(* CODESYS project TcNexaHmi.library
   Author: ATI Software Engineering
   Version: 2.0.0
   Title: TcNexaHmi
   DefaultNamespace: TcNexa_Devices_Hmi_TcNexaHmi
   Placeholder: TcNexaHmi
   Company: TcNexa

Project tree, tasks and I/O mapping:
  libraries: Tc2_Standard, * (Beckhoff Automation GmbH); Tc2_System, * (Beckhoff Automation GmbH); Tc2_Utilities, * (Beckhoff Automation GmbH); Tc3_IotBase, * (Beckhoff Automation GmbH); Tc3_Module, * (Beckhoff Automation GmbH); TcUtilities, * (TcNexa)
  Base/
    ITFs/
      interface I_NexaHmi: isConnected, messageFullTopic, messageLastTopicLevel, messagePayload, onNewMessage, publish, publishAdr, subscribe, topicPrefix, unsubscribe
    POUs/
      function block FB_NexaHmi [ST]: hostName, hostPort, id, isConnected, messageFullTopic, messageLastTopicLevel, messagePayload, onNewMessage, topicPrefix, FB_main, publish, publishAdr, setWill, subscribe, unsubscribe
    data type E_UserLevel
    function F_GetUserLevelAsString [ST]
  Device Buttons/
    function block FB_NexaHmiDeviceButton [ST]: _handleNewMessages, _onConnection, _updateTopics, FB_init, Buttons, description, FB_main
  Elements/
    Counters/
      data type E_NexaHmiCounterColor
      function block FB_NexaHmiCounter [ST]: color, description, name, value, _getColor, _handleNewMessages, _onConnection, _updateTopics, clear, FB_init, FB_main, inc
    Graph 2D/
      data type E_GraphLineColor2D
      function block FB_NexaHmi_Graph2D [ST]: _onConnection, _updateTopics, FB_init, description, Lines, xMax, xMaxVisible, xMin, xMinVisible, yMax, yMaxVisible, yMin, yMinVisible, clear, FB_main, publish
      function block FB_NexaHmi_GraphLine2D [ST]: _clearBuffer, _getColor, _onConnection, _updateTopics, Hmi, topicPrefix, addPoint, clear, FB_main, publish, setColor
    POUs/
      function block FB_CustomHmiButton [ST]: focused, name, onTap, visible, clear
      function block FB_GeneralHmiButton [ST]: confirmationRequired, enabled, focused, isPressed, loggingEnabled, name, onTap, visible, clear
      function block FB_ModeHmiButton [ST]: enabled, onLongPress, onTap, visible, clear, clearCommand
      function block FB_NexaHmiCustomButtons [ST]: Buttons, clear
      function block FB_NexaHmiTextFields [ST]: fields, userAction, clear
  GVLs/
    global variables GVL_TcNexaHmiUtilities
  Order/
    function block FB_NexaHmiOrderBOOL [ST]: _handleNewMessages, _onConnection, _updateTopics, FB_init, description, name, value, FB_main
    function block FB_NexaHmiOrderINT [ST]: _handleNewMessage, _onConnection, _updateTopics, FB_init, description, lowerLimit, name, upperLimit, value, FB_main
    function block FB_NexaHmiOrderREAL [ST]: _handleNewMessage, _onConnection, _updateTopics, FB_init, description, lowerLimit, name, upperLimit, value, FB_main
    function block FB_NexaHmiOrderSTRING [ST]: _handleNewMessages, _onConnection, _updateTopics, FB_init, value, FB_main
    function block FB_NexaHmiOrderTIME [ST]: _handleNewMessages, _onConnection, _updateTopics, FB_init, description, name, value, FB_main
  Persistent/
    function block FB_NexaHmiPersistentBase [ST]: _handleVar, _onConnection, FB_init, FB_main
    function block FB_NexaHmiPersistentBOOL [ST]: _handleVar, FB_init, value
    function block FB_NexaHmiPersistentINT [ST]: _handleVar, FB_init, value
    function block FB_NexaHmiPersistentREAL [ST]: _handleVar, FB_init, value
    function block FB_NexaHmiPersistentSTRING [ST]: _handleVar, FB_init, value
    function block FB_NexaHmiPersistentTIME [ST]: _handleVar, FB_init, value
    function block FB_NexaHmiPersistentXYZ [ST]: _handleVar, FB_init, velocity, X, Y, Z
  Settings/
    function block FB_NexaHmiSettingBase [ST]: _handleVars, _onConnection, _updateTopics, FB_init, description, enabled, name, userLevel, FB_main
    function block FB_NexaHmiSettingBOOL [ST]: _handleVars, FB_init, value
    function block FB_NexaHmiSettingCHOICE [ST]: _handleVars, FB_init, value
    function block FB_NexaHmiSettingINT [ST]: _handleVars, FB_init, lowerLimit, upperLimit, value
    function block FB_NexaHmiSettingREAL [ST]: _handleVars, FB_init, lowerLimit, upperLimit, value
    function block FB_NexaHmiSettingSTRING [ST]: _handleVars, FB_init, value
    function block FB_NexaHmiSettingTIME [ST]: _handleVars, FB_init, lowerLimit, upperLimit, value
  Tests/
    program PRG_TEST [ST]
  Version/
    global variables Global_Version
*)

// Base/E_UserLevel
{attribute 'qualified_only'}
{attribute 'strict'}
TYPE E_UserLevel :
(
	Operator := 0,
	LineLeader,
	Maintenance,
	Administrator,
	System
):= Administrator;
END_TYPE

// Elements/Counters/E_NexaHmiCounterColor
{attribute 'qualified_only'}
{attribute 'strict'}
TYPE E_NexaHmiCounterColor :
(
	black := 0,
	red,
	blue,
	green,
	yellow,
	purple,
	grey
):= black;
END_TYPE

// Elements/Graph 2D/E_GraphLineColor2D
{attribute 'qualified_only'}
{attribute 'strict'}
TYPE E_GraphLineColor2D :
(
	black := 0,
	red,
	blue,
	green,
	yellow,
	purple,
	grey
):= black;
END_TYPE

// GVLs/GVL_TcNexaHmiUtilities
{attribute 'qualified_only'}
VAR_GLOBAL CONSTANT
	numOfTextFields			: USINT:= 3;
	numOfCustomButtons		: USINT:= 5;
	numOfGraphLines2D		: USINT:= 5;
END_VAR

// Version/Global_Version
{attribute 'TcGenerated'}
{attribute 'no-analysis'}
{attribute 'linkalways'}
// This function has been automatically generated from the project information.
VAR_GLOBAL CONSTANT
	{attribute 'const_non_replaced'}
	stLibVersion_TcNexaHmi : ST_LibVersion := (iMajor := 2, iMinor := 0, iBuild := 0, iRevision := 0, nFlags := 0, sVersion := '2.0.0');
END_VAR

// Base/ITFs/I_NexaHmi
INTERFACE I_NexaHmi

PROPERTY PUBLIC isConnected : BOOL
GET
END_GET
END_PROPERTY

PROPERTY messageFullTopic : Tc2_System.T_MaxString
GET
END_GET
END_PROPERTY

PROPERTY PUBLIC messageLastTopicLevel : STRING
GET
END_GET
END_PROPERTY

PROPERTY messagePayload : Tc2_System.T_MaxString
GET
END_GET
END_PROPERTY

PROPERTY PUBLIC onNewMessage : BOOL
GET
END_GET
END_PROPERTY

METHOD PUBLIC publish : BOOL
VAR_INPUT
	topic		: Tc2_System.T_MaxString;
	payload		: Tc2_System.T_MaxString;
END_VAR
END_METHOD

METHOD PUBLIC publishAdr : BOOL
VAR_INPUT
	topic		: Tc2_System.T_MaxString;
	payload		: PVOID;
	payloadSize	: UDINT;
END_VAR
END_METHOD

METHOD PUBLIC subscribe : BOOL
VAR_INPUT
	topic		: Tc2_System.T_MaxString;
END_VAR
END_METHOD

PROPERTY PUBLIC topicPrefix : Tc2_System.T_MaxString
GET
END_GET
END_PROPERTY

METHOD PUBLIC unsubscribe
VAR_INPUT
	topic		: Tc2_System.T_MaxString;
END_VAR
END_METHOD

END_INTERFACE

// Base/POUs/FB_NexaHmi
FUNCTION_BLOCK FB_NexaHmi IMPLEMENTS I_NexaHmi
VAR
	(* Mqtt *)
	_Client						: Tc3_IotBase.FB_IotMqttClient;
	_ClientMessageQueue			: Tc3_IotBase.FB_IotMqttMessageQueue;
	_ClientMessage				: Tc3_IotBase.FB_IotMqttMessage;
	_isInit						: BOOL;
	_onNewMessage				: BOOL;
	_topicPrefix				: Tc2_System.T_MaxString;
	(* Message *)
	_messageTopic				: Tc2_System.T_MaxString;
	_messageTopicSplitter		: TcNexa_Components_TcUtilities.FB_TextSplitter;
	_messagePayload				: Tc2_System.T_MaxString;
	(* Will *)
	_willTopic					: STRING;
	_willPayload				: STRING;
END_VAR

PROPERTY PUBLIC hostName : Tc2_System.T_MaxString
GET
hostName:= _Client.sHostName;
END_GET
SET
_Client.sHostName:= hostName;
END_SET
END_PROPERTY

PROPERTY PUBLIC hostPort : UINT
GET
hostPort:= _Client.nHostPort;
END_GET
SET
_Client.nHostPort:= hostPort;
END_SET
END_PROPERTY

PROPERTY PUBLIC id : Tc2_System.T_MaxString
GET
id:= _Client.sClientId;
END_GET
SET
_Client.sClientId:= id;
END_SET
END_PROPERTY

PROPERTY PUBLIC isConnected : BOOL
GET
isConnected:= _Client.bConnected;
END_GET
END_PROPERTY

PROPERTY messageFullTopic : Tc2_System.T_MaxString
GET
messageFullTopic:= _messageTopic;
END_GET
END_PROPERTY

PROPERTY PUBLIC messageLastTopicLevel : STRING
GET
messageLastTopicLevel:= _messageTopicSplitter.getValueAt(index:= _messageTopicSplitter.size, Response:= 0);
END_GET
END_PROPERTY

PROPERTY messagePayload : Tc2_System.T_MaxString
GET
messagePayload:= _messagePayload;
END_GET
END_PROPERTY

PROPERTY PUBLIC onNewMessage : BOOL
GET
onNewMessage:= _onNewMessage;
END_GET
END_PROPERTY

PROPERTY PUBLIC topicPrefix : Tc2_System.T_MaxString
GET
topicPrefix:= _topicPrefix;
END_GET
SET
_topicPrefix:= topicPrefix;
END_SET
END_PROPERTY

METHOD PUBLIC FB_main
VAR_INPUT
END_VAR
IF NOT _isInit THEN
	_Client.ipMessageQueue:= _ClientMessageQueue;
	_isInit:= TRUE;
END_IF
_Client.Execute(bConnect:= TRUE);

_onNewMessage:= FALSE;
IF (_ClientMessageQueue.nQueuedMessages > 0) THEN
	IF _ClientMessageQueue.Dequeue(fbMessage:= _ClientMessage)  THEN
		_ClientMessage.GetTopic(
			pTopic				:= ADR(_messageTopic),
			nTopicSize			:= SIZEOF(_messageTopic));
		_ClientMessage.GetPayload(
			pPayload			:= ADR(_messagePayload),
			nPayloadSize		:= SIZEOF(_messagePayload),
			bSetNullTermination	:= TRUE);
		_messageTopicSplitter.split(
			source				:= _messageTopic,
			delimiter			:= '/',
			Response			:= 0);
		_onNewMessage:= TRUE;
	END_IF
ELSE
	_messageTopic:= '';
	_messagePayload:= '';
END_IF
END_METHOD

METHOD PUBLIC publish : BOOL
VAR_INPUT
	topic		: Tc2_System.T_MaxString;
	payload		: Tc2_System.T_MaxString;
END_VAR
publish:= _Client.Publish(
			sTopic			:= topic,
			pPayload		:= ADR(payload),
			nPayloadSize	:= INT_TO_UDINT(Tc2_Standard.LEN(payload)),
			eQoS			:= TcIotMqttQos.AtMostOnceDelivery,
			bRetain			:= TRUE,
			bQueue			:= FALSE);
END_METHOD

METHOD PUBLIC publishAdr : BOOL
VAR_INPUT
	topic		: Tc2_System.T_MaxString;
	payload		: PVOID;
	payloadSize	: UDINT;
END_VAR
publishAdr:= _Client.Publish(
			sTopic			:= topic,
			pPayload		:= payload,
			nPayloadSize	:= payloadSize,
			eQoS			:= TcIotMqttQos.AtMostOnceDelivery,
			bRetain			:= TRUE,
			bQueue			:= FALSE);
END_METHOD

METHOD PUBLIC setWill
VAR_INPUT
	topic		: Tc2_System.T_MaxString;
	payload		: Tc2_System.T_MaxString;
END_VAR
_willTopic:= topic;
THIS^._willPayload:= payload;
THIS^._Client.stWill.sTopic:= _willTopic;
THIS^._Client.stWill.pPayload:= ADR(_willPayload);
THIS^._Client.stWill.nPayloadSize:= INT_TO_UDINT(Tc2_Standard.LEN(_willPayload));
THIS^._Client.stWill.eQoS:= TcIotMqttQos.AtMostOnceDelivery;
THIS^._Client.stWill.bRetain:= TRUE;
END_METHOD

METHOD PUBLIC subscribe : BOOL
VAR_INPUT
	topic		: Tc2_System.T_MaxString;
END_VAR
subscribe:= _Client.Subscribe(
				sTopic	:= topic,
				eQoS	:= TcIotMqttQos.AtLeastOnceDelivery);
END_METHOD

METHOD PUBLIC unsubscribe
VAR_INPUT
	topic		: Tc2_System.T_MaxString;
END_VAR
_Client.Unsubscribe(sTopic:= topic);
END_METHOD

END_FUNCTION_BLOCK

// Base/F_GetUserLevelAsString
FUNCTION F_GetUserLevelAsString : STRING
VAR_INPUT
	userLevel		: E_UserLevel;
END_VAR
VAR
END_VAR

IF (userLevel = E_UserLevel.Operator) THEN
	F_GetUserLevelAsString:= 'operator';
ELSIF (userLevel = E_UserLevel.LineLeader) THEN
	F_GetUserLevelAsString:= 'lineLeader';
ELSIF (userLevel = E_UserLevel.Maintenance) THEN
	F_GetUserLevelAsString:= 'maintenance';
ELSIF (userLevel = E_UserLevel.Administrator) THEN
	F_GetUserLevelAsString:= 'admin';
ELSIF (userLevel = E_UserLevel.System) THEN
	F_GetUserLevelAsString:= 'system';
END_IF

END_FUNCTION

// Device Buttons/FB_NexaHmiDeviceButton
FUNCTION_BLOCK FB_NexaHmiDeviceButton
VAR
	_Hmi				: I_NexaHmi;
	_timerConnected		: Tc2_Standard.TON;
	_onHmiConnection	: Tc2_Standard.R_TRIG;
	_isHmiConnected		: BOOL;
	_topicPrefix		: Tc2_System.T_MaxString;
	_id					: UINT;
	_name				: Tc2_System.T_MaxString;
	_description		: Tc2_System.T_MaxString;
	_Buttons			: ARRAY[1..NUM_OF_BUTTONS] OF FB_GeneralHmiButton;
	_LastButtons		: ARRAY[1..NUM_OF_BUTTONS] OF FB_GeneralHmiButton;
	_lastDescription	: Tc2_System.T_MaxString;		
	_tmpCounter			: USINT;
	_tmpText			: Tc2_System.T_MaxString;
END_VAR
VAR CONSTANT
	NUM_OF_BUTTONS		: USINT:= 3;
END_VAR

METHOD PROTECTED _handleNewMessages
VAR_INPUT
END_VAR
IF NOT _isHmiConnected THEN RETURN; END_IF

IF _Hmi.onNewMessage THEN
	FOR _tmpCounter:= 1 TO NUM_OF_BUTTONS DO
		_tmpText:= Tc2_Standard.CONCAT(STR1:= _topicPrefix, STR2:= 'buttons/');
		_tmpText:= Tc2_Standard.CONCAT(STR1:= _tmpText, STR2:= USINT_TO_STRING(_tmpCounter));
		_tmpText:= Tc2_Standard.CONCAT(STR1:= _tmpText, STR2:= '/action');
		IF (_Hmi.messageFullTopic = _tmpText) THEN
			IF (_Hmi.messagePayload = 'tap') AND _Buttons[_tmpCounter].enabled THEN
				_Buttons[_tmpCounter].onTap:= TRUE;
// 			ELSIF (_Hmi.messagePayload = 'longPress') AND _Buttons[_tmpCounter].enabled THEN
// 				_Buttons[_tmpCounter].isPressed:= TRUE;
			END_IF
		END_IF
	END_FOR
END_IF
END_METHOD

METHOD PROTECTED _onConnection
VAR_INPUT
END_VAR
IF NOT _onHmiConnection.Q THEN RETURN; END_IF

_topicPrefix:= Tc2_Standard.CONCAT(STR1:= _Hmi.topicPrefix, STR2:= 'devices/buttons/');
_topicPrefix:= Tc2_Standard.CONCAT(STR1:= _topicPrefix, STR2:= UINT_TO_STRING(_id));
_topicPrefix:= Tc2_Standard.CONCAT(STR1:= _topicPrefix, STR2:= '/');

FOR _tmpCounter:= 1 TO NUM_OF_BUTTONS DO
	_tmpText:= CONCAT(STR1:= _topicPrefix, STR2:= 'buttons/');
	_tmpText:= CONCAT(STR1:= _tmpText, STR2:= USINT_TO_STRING(_tmpCounter));
	_tmpText:= CONCAT(STR1:= _tmpText, STR2:= '/action');
	_Hmi.subscribe(topic:= _tmpText);
END_FOR

_Hmi.publish(
	topic	:= Tc2_Standard.CONCAT(STR1:= _topicPrefix, STR2:= 'active'),
	payload	:= BOOL_TO_STRING(TRUE));
_Hmi.publish(
	topic	:= Tc2_Standard.CONCAT(STR1:= _topicPrefix, STR2:= 'name'),
	payload	:= _name);
END_METHOD

METHOD PROTECTED _updateTopics
VAR_INPUT
END_VAR
IF NOT _isHmiConnected THEN RETURN; END_IF

(* Description *)
IF (_lastDescription <> _description) OR _onHmiConnection.Q THEN
	_lastDescription:= _description;
	_Hmi.publish(
		topic	:= Tc2_Standard.CONCAT(STR1:= _topicPrefix, STR2:= 'description'),
		payload	:= _description);
END_IF
(* Handle Buttons *)
FOR _tmpCounter:= 1 TO NUM_OF_BUTTONS DO
	(* Button Name *)
	IF (_LastButtons[_tmpCounter].name <> _Buttons[_tmpCounter].name) OR _onHmiConnection.Q THEN
		_LastButtons[_tmpCounter].name:= _Buttons[_tmpCounter].name;
		_tmpText:= Tc2_Standard.CONCAT(STR1:= _topicPrefix, STR2:= 'buttons/');
		_tmpText:= Tc2_Standard.CONCAT(STR1:= _tmpText, STR2:= USINT_TO_STRING(_tmpCounter));
		_tmpText:= Tc2_Standard.CONCAT(STR1:= _tmpText, STR2:= '/name');
		_Hmi.publish(
			topic	:= _tmpText,
			payload	:= _Buttons[_tmpCounter].name);
	END_IF
	(* Button Visible *)
	IF (_LastButtons[_tmpCounter].visible <> _Buttons[_tmpCounter].visible) OR _onHmiConnection.Q THEN
		_LastButtons[_tmpCounter].visible:= _Buttons[_tmpCounter].visible;
		_tmpText:= Tc2_Standard.CONCAT(STR1:= _topicPrefix, STR2:= 'buttons/');
		_tmpText:= Tc2_Standard.CONCAT(STR1:= _tmpText, STR2:= USINT_TO_STRING(_tmpCounter));
		_tmpText:= Tc2_Standard.CONCAT(STR1:= _tmpText, STR2:= '/visible');
		_Hmi.publish(
			topic	:= _tmpText,
			payload	:= BOOL_TO_STRING(_Buttons[_tmpCounter].visible));
	END_IF
	(* Button Enabled *)
	IF (_LastButtons[_tmpCounter].enabled <> _Buttons[_tmpCounter].enabled) OR _onHmiConnection.Q THEN
		_LastButtons[_tmpCounter].enabled:= _Buttons[_tmpCounter].enabled;
		_tmpText:= Tc2_Standard.CONCAT(STR1:= _topicPrefix, STR2:= 'buttons/');
		_tmpText:= Tc2_Standard.CONCAT(STR1:= _tmpText, STR2:= USINT_TO_STRING(_tmpCounter));
		_tmpText:= Tc2_Standard.CONCAT(STR1:= _tmpText, STR2:= '/enabled');
		_Hmi.publish(
			topic	:= _tmpText,
			payload	:= BOOL_TO_STRING(_Buttons[_tmpCounter].enabled));
	END_IF
	(* Button Focused *)
	IF (_LastButtons[_tmpCounter].focused <> _Buttons[_tmpCounter].focused) OR _onHmiConnection.Q THEN
		_LastButtons[_tmpCounter].focused:= _Buttons[_tmpCounter].focused;
		_tmpText:= Tc2_Standard.CONCAT(STR1:= _topicPrefix, STR2:= 'buttons/');
		_tmpText:= Tc2_Standard.CONCAT(STR1:= _tmpText, STR2:= USINT_TO_STRING(_tmpCounter));
		_tmpText:= Tc2_Standard.CONCAT(STR1:= _tmpText, STR2:= '/focused');
		_Hmi.publish(
			topic	:= _tmpText,
			payload	:= BOOL_TO_STRING(_Buttons[_tmpCounter].focused));
	END_IF	
	(* Button Confirmation *)
	IF (_LastButtons[_tmpCounter].confirmationRequired <> _Buttons[_tmpCounter].confirmationRequired) OR _onHmiConnection.Q THEN
		_LastButtons[_tmpCounter].confirmationRequired:= _Buttons[_tmpCounter].confirmationRequired;
		_tmpText:= Tc2_Standard.CONCAT(STR1:= _topicPrefix, STR2:= 'buttons/');
		_tmpText:= Tc2_Standard.CONCAT(STR1:= _tmpText, STR2:= USINT_TO_STRING(_tmpCounter));
		_tmpText:= Tc2_Standard.CONCAT(STR1:= _tmpText, STR2:= '/confirmationRequired');
		_Hmi.publish(
			topic	:= _tmpText,
			payload	:= BOOL_TO_STRING(_Buttons[_tmpCounter].confirmationRequired));
	END_IF	
	(* Button Confirmation *)
	IF (_LastButtons[_tmpCounter].loggingEnabled <> _Buttons[_tmpCounter].loggingEnabled) OR _onHmiConnection.Q THEN
		_LastButtons[_tmpCounter].loggingEnabled:= _Buttons[_tmpCounter].loggingEnabled;
		_tmpText:= Tc2_Standard.CONCAT(STR1:= _topicPrefix, STR2:= 'buttons/');
		_tmpText:= Tc2_Standard.CONCAT(STR1:= _tmpText, STR2:= USINT_TO_STRING(_tmpCounter));
		_tmpText:= Tc2_Standard.CONCAT(STR1:= _tmpText, STR2:= '/loggingEnabled');
		_Hmi.publish(
			topic	:= _tmpText,
			payload	:= BOOL_TO_STRING(_Buttons[_tmpCounter].loggingEnabled));
	END_IF	
	
	_Buttons[_tmpCounter].onTap:= FALSE;
	_Buttons[_tmpCounter].isPressed:= FALSE;
END_FOR
END_METHOD

METHOD FB_init : BOOL
VAR_INPUT
	bInitRetains	: BOOL; // if TRUE, the retain variables are initialized (warm start / cold start)
	bInCopyCode 	: BOOL;  // if TRUE, the instance afterwards gets moved into the copy code (online change)
	Hmi				: I_NexaHmi;
	id				: UINT;
	name			: Tc2_System.T_MaxString;
	descrpiton		: Tc2_System.T_MaxString;
END_VAR
THIS^._Hmi:= Hmi;
THIS^._id:= id;
THIS^._name:= name;
THIS^._description:= descrpiton;
END_METHOD

PROPERTY Buttons : REFERENCE TO ARRAY[1..NUM_OF_BUTTONS] OF FB_GeneralHmiButton
GET
Buttons REF= _Buttons;
END_GET
END_PROPERTY

PROPERTY description : Tc2_System.T_MaxString
GET
description:= _description;
END_GET
SET
_description:= description;
END_SET
END_PROPERTY

METHOD PUBLIC FB_main
VAR_INPUT
END_VAR
_timerConnected(IN:= _Hmi.isConnected, PT:= T#1S);
_isHmiConnected:= _timerConnected.Q;
_onHmiConnection(CLK:= _isHmiConnected);

_onConnection();
_updateTopics();
_handleNewMessages();
END_METHOD

END_FUNCTION_BLOCK

// Elements/POUs/FB_GeneralHmiButton
FUNCTION_BLOCK FB_GeneralHmiButton
VAR
	_name						: STRING;
	_visible					: BOOL;
	_enabled					: BOOL;
	_focused					: BOOL;
	_onTap						: BOOL;
	_isPressed					: BOOL;
	_confirmationRequired		: BOOL;
	_loggingEnabled				: BOOL;
END_VAR

PROPERTY confirmationRequired : BOOL
GET
confirmationRequired:= _confirmationRequired;
END_GET
SET
_confirmationRequired:= confirmationRequired;
END_SET
END_PROPERTY

PROPERTY PUBLIC enabled : BOOL
GET
enabled:= _enabled;
END_GET
SET
_enabled:= enabled;
END_SET
END_PROPERTY

PROPERTY PUBLIC focused : BOOL
GET
focused:= _focused;
END_GET
SET
_focused:= focused;
END_SET
END_PROPERTY

PROPERTY PUBLIC isPressed : BOOL
GET
isPressed:= _isPressed;
END_GET
SET
_isPressed:= isPressed;
END_SET
END_PROPERTY

PROPERTY loggingEnabled : BOOL
GET
loggingEnabled:= _loggingEnabled;
END_GET
SET
_loggingEnabled:= loggingEnabled;
END_SET
END_PROPERTY

PROPERTY PUBLIC name : STRING
GET
name:= _name;
END_GET
SET
_name:= name;
END_SET
END_PROPERTY

PROPERTY PUBLIC onTap : BOOL
GET
onTap:= _onTap;
END_GET
SET
_onTap:= onTap;
END_SET
END_PROPERTY

PROPERTY PUBLIC visible : BOOL
GET
visible:= _visible;
END_GET
SET
_visible:= visible;
END_SET
END_PROPERTY

METHOD PUBLIC clear
VAR_INPUT
END_VAR
_name:= '';
_confirmationRequired:= FALSE;
_focused:= FALSE;
_enabled:= FALSE;
END_METHOD

END_FUNCTION_BLOCK

// Elements/Counters/FB_NexaHmiCounter
FUNCTION_BLOCK FB_NexaHmiCounter
VAR
	_Hmi				: I_NexaHmi;
	_onHmiConnection	: Tc2_Standard.R_TRIG;
	_isHmiConnected		: BOOL;
	_id					: STRING;
	_name				: STRING(255);
	_description		: STRING(255);
	_value				: UDINT;
	_color				: E_NexaHmiCounterColor;
	(* General *)
	_timerPublish		: Tc2_Standard.TON;
	_topicPrefix		: Tc2_System.T_MaxString;
	(* Last values *)
	_lastDescription	: STRING(255);
	_lastValue			: UDINT;
	_lastColor			: E_NexaHmiCounterColor;
END_VAR

PROPERTY color : E_NexaHmiCounterColor
GET
color:= _color;
END_GET
SET
_color:= color;
END_SET
END_PROPERTY

PROPERTY description : Tc2_System.T_MaxString
GET
description:= _description;
END_GET
END_PROPERTY

PROPERTY name : Tc2_System.T_MaxString
GET
name:= _name;
END_GET
END_PROPERTY

PROPERTY PUBLIC value : UDINT
GET
value:= _value;
END_GET
END_PROPERTY

METHOD PROTECTED _getColor : STRING
VAR_INPUT
END_VAR
IF (_color = E_NexaHmiCounterColor.black) THEN
	_getColor:= 'black';
ELSIF (_color = E_NexaHmiCounterColor.blue) THEN
	_getColor:= 'blue';
ELSIF (_color = E_NexaHmiCounterColor.green) THEN
	_getColor:= 'green';
ELSIF (_color = E_NexaHmiCounterColor.grey) THEN
	_getColor:= 'grey';
ELSIF (_color = E_NexaHmiCounterColor.purple) THEN
	_getColor:= 'purple';
ELSIF (_color = E_NexaHmiCounterColor.red) THEN
	_getColor:= 'red';
ELSIF (_color = E_NexaHmiCounterColor.yellow) THEN
	_getColor:= 'yellow';
END_IF
END_METHOD

METHOD PROTECTED _handleNewMessages
VAR_INPUT
END_VAR
IF NOT _isHmiConnected THEN RETURN; END_IF

IF _Hmi.onNewMessage THEN
	IF (Tc2_Standard.FIND(STR1:= _Hmi.messageFullTopic, STR2:= _topicPrefix) <> 0) THEN
		IF (_Hmi.messageFullTopic = Tc2_Standard.CONCAT(STR1:= _topicPrefix, STR2:= 'value')) THEN
			_value:= STRING_TO_UDINT(_Hmi.messagePayload);
			_lastValue:= _value;
		END_IF
	END_IF
END_IF
END_METHOD

METHOD PROTECTED _onConnection
VAR_INPUT
END_VAR
IF NOT _onHmiConnection.Q THEN RETURN; END_IF

_topicPrefix:= Tc2_Standard.CONCAT(STR1:= _Hmi.topicPrefix, STR2:= 'overview/counters/');
// _topicPrefix:= Tc2_Standard.CONCAT(STR1:= _topicPrefix, STR2:= UINT_TO_STRING(_id));
_topicPrefix:= Tc2_Standard.CONCAT(STR1:= _topicPrefix, STR2:= _id);
_topicPrefix:= Tc2_Standard.CONCAT(STR1:= _topicPrefix, STR2:= '/');

_Hmi.subscribe(topic:= Tc2_Standard.CONCAT(STR1:= _topicPrefix, STR2:= 'value'));

_Hmi.publish(
	topic	:= Tc2_Standard.CONCAT(STR1:= _topicPrefix, STR2:= 'active'),
	payload	:= BOOL_TO_STRING(TRUE));
_Hmi.publish(
	topic	:= Tc2_Standard.CONCAT(STR1:= _topicPrefix, STR2:= 'name'),
	payload	:= _name);
END_METHOD

METHOD PROTECTED _updateTopics
VAR_INPUT
END_VAR
IF NOT _isHmiConnected THEN RETURN; END_IF

(* Value *)
IF (_lastValue <> _value) AND _timerPublish.Q THEN
	_lastValue:= _value;
	_Hmi.publish(
		topic	:= Tc2_Standard.CONCAT(STR1:= _topicPrefix, STR2:= 'value'),
		payload	:= UDINT_TO_STRING(_value));
END_IF
(* Enabled *)
IF (_lastDescription <> _description) OR _onHmiConnection.Q THEN
	_lastDescription:= _description;
	_Hmi.publish(
		topic	:= Tc2_Standard.CONCAT(STR1:= _topicPrefix, STR2:= 'description'),
		payload	:= _description);
END_IF
(* Color *)
IF (_lastColor <> _color) OR _onHmiConnection.Q THEN
	_lastColor:= _color;
	_Hmi.publish(
		topic	:= Tc2_Standard.CONCAT(STR1:= _topicPrefix, STR2:= 'color'),
		payload	:= _getColor());
END_IF
END_METHOD

METHOD clear
VAR_INPUT
END_VAR
_value:= 0;
END_METHOD

METHOD FB_init : BOOL
VAR_INPUT
	bInitRetains	: BOOL; // if TRUE, the retain variables are initialized (warm start / cold start)
	bInCopyCode 	: BOOL;  // if TRUE, the instance afterwards gets moved into the copy code (online change)
	Hmi				: I_NexaHmi;
	id				: STRING(39);
	name			: STRING(255);
END_VAR
VAR
	_temp			: INT;
END_VAR
THIS^._Hmi:= Hmi;
THIS^._id:= id;
THIS^._name:= name;
END_METHOD

METHOD PUBLIC FB_main
VAR_INPUT
END_VAR
_timerPublish(
	IN:= _isHmiConnected, 
	PT:= T#1S);
_isHmiConnected:= _Hmi.isConnected;
_onHmiConnection(
	CLK:= _isHmiConnected);

_onConnection();
_updateTopics();
_handleNewMessages();
END_METHOD

METHOD PUBLIC inc
VAR_INPUT
END_VAR
_value:= _value + 1;
END_METHOD

END_FUNCTION_BLOCK

// Elements/Graph 2D/FB_NexaHmi_Graph2D
FUNCTION_BLOCK FB_NexaHmi_Graph2D
VAR
	_Hmi				: I_NexaHmi;
	_onHmiConnection	: Tc2_Standard.R_TRIG;
	_isHmiConnected		: BOOL;
	_topicPrefix		: Tc2_System.T_MaxString;
	_id					: Tc2_System.T_MaxString;
	_name				: Tc2_System.T_MaxString;
	_description		: Tc2_System.T_MaxString;
	_xTitle				: STRING;
	_xMin				: REAL;
	_xMinVisible		: BOOL;
	_xMax				: REAL;
	_xMaxVisible		: BOOL;
	_yTitle				: STRING;
	_yMin				: REAL;
	_yMinVisible		: BOOL;
	_yMax				: REAL;
	_yMaxVisible		: BOOL;
	_tmpText			: Tc2_System.T_MaxString;
	_counter			: USINT;
	_Lines				: ARRAY[1..GVL_TcNexaHmiUtilities.numOfGraphLines2D] OF FB_NexaHmi_GraphLine2D;
	(* *)
	_lastDescription	: Tc2_System.T_MaxString;
	_xLastMin			: REAL;
	_xLastMinVisible	: BOOL;
	_xLastMax			: REAL;
	_xLastMaxVisible	: BOOL;
	_yLastMin			: REAL;
	_yLastMinVisible	: BOOL;
	_yLastMax			: REAL;
	_yLastMaxVisible	: BOOL;
END_VAR

METHOD PROTECTED _onConnection
VAR_INPUT
END_VAR
IF NOT _onHmiConnection.Q THEN RETURN; END_IF

_topicPrefix:= Tc2_Standard.CONCAT(STR1:= _Hmi.topicPrefix, STR2:= 'overview/graphs2d/');
_topicPrefix:= Tc2_Standard.CONCAT(STR1:= _topicPrefix, STR2:= _id);
_topicPrefix:= Tc2_Standard.CONCAT(STR1:= _topicPrefix, STR2:= '/');

_Hmi.publish(
	topic	:= Tc2_Standard.CONCAT(STR1:= _topicPrefix, STR2:= 'active'),
	payload	:= BOOL_TO_STRING(TRUE));
_Hmi.publish(
	topic	:= Tc2_Standard.CONCAT(STR1:= _topicPrefix, STR2:= 'general/name'),
	payload	:= _name);
_Hmi.publish(
	topic	:= Tc2_Standard.CONCAT(STR1:= _topicPrefix, STR2:= 'general/xAxisTitle'),
	payload	:= _xTitle);
_Hmi.publish(
	topic	:= Tc2_Standard.CONCAT(STR1:= _topicPrefix, STR2:= 'general/yAxisTitle'),
	payload	:= _yTitle);
	
FOR _counter:= 1 TO GVL_TcNexaHmiUtilities.numOfGraphLines2D DO
	_tmpText:= Tc2_Standard.CONCAT(STR1:= _topicPrefix, STR2:= 'lines/');
	_tmpText:= Tc2_Standard.CONCAT(STR1:= _tmpText, STR2:= USINT_TO_STRING(_counter));
	_tmpText:= Tc2_Standard.CONCAT(STR1:= _tmpText, STR2:= '/');
	_Lines[_counter].topicPrefix:= _tmpText;
END_FOR
END_METHOD

METHOD PROTECTED _updateTopics
VAR_INPUT
END_VAR
IF NOT _isHmiConnected THEN RETURN; END_IF

(* Description *)
IF (_lastDescription <> _description) OR _onHmiConnection.Q THEN
	_lastDescription:= _description;
	_Hmi.publish(
		topic	:= Tc2_Standard.CONCAT(STR1:= _topicPrefix, STR2:= 'general/description'),
		payload	:= _description);	
END_IF
(* X Min *)
IF ((_xLastMin <> _xMin) OR _onHmiConnection.Q) THEN
	_xLastMin:= _xMin;
	IF NOT _xMinVisible THEN
		_Hmi.publish(
			topic	:= Tc2_Standard.CONCAT(STR1:= _topicPrefix, STR2:= 'general/xAxisMin'),
			payload	:= '');	
	ELSE
		_Hmi.publish(
			topic	:= Tc2_Standard.CONCAT(STR1:= _topicPrefix, STR2:= 'general/xAxisMin'),
			payload	:= REAL_TO_STRING(_xMin));		
	END_IF
END_IF
(* X Min Visible *)
IF (_xLastMinVisible <> _xMinVisible) OR _onHmiConnection.Q THEN
	_xLastMinVisible:= _xMinVisible;
	_xLastMin:= _xMin;
	IF NOT _xMinVisible THEN
		_Hmi.publish(
			topic	:= Tc2_Standard.CONCAT(STR1:= _topicPrefix, STR2:= 'general/xAxisMin'),
			payload	:= '');	
	ELSE
		_Hmi.publish(
			topic	:= Tc2_Standard.CONCAT(STR1:= _topicPrefix, STR2:= 'general/xAxisMin'),
			payload	:= REAL_TO_STRING(_xMin));		
	END_IF
END_IF
(* X Max *)
IF ((_xLastMax <> _xMax) OR _onHmiConnection.Q) THEN
	_xLastMax:= _xMax;
	IF NOT _xMaxVisible THEN
		_Hmi.publish(
			topic	:= Tc2_Standard.CONCAT(STR1:= _topicPrefix, STR2:= 'general/xAxisMax'),
			payload	:= '');		
	ELSE
		_Hmi.publish(
			topic	:= Tc2_Standard.CONCAT(STR1:= _topicPrefix, STR2:= 'general/xAxisMax'),
			payload	:= REAL_TO_STRING(_xMax));	
	END_IF
END_IF
(* X Max Visible *)
IF (_xLastMaxVisible <> _xMaxVisible) OR _onHmiConnection.Q THEN
	_xLastMaxVisible:= _xMaxVisible;
	_xLastMax:= _xMax;
	IF NOT _xMaxVisible THEN
		_Hmi.publish(
			topic	:= Tc2_Standard.CONCAT(STR1:= _topicPrefix, STR2:= 'general/xAxisMax'),
			payload	:= '');		
	ELSE
		_Hmi.publish(
			topic	:= Tc2_Standard.CONCAT(STR1:= _topicPrefix, STR2:= 'general/xAxisMax'),
			payload	:= REAL_TO_STRING(_xMax));	
	END_IF
END_IF
(* Y Min *)
IF ((_yLastMin <> _yMin) OR _onHmiConnection.Q) THEN
	_yLastMin:= _yMin;
	IF NOT _yMinVisible THEN
		_Hmi.publish(
			topic	:= Tc2_Standard.CONCAT(STR1:= _topicPrefix, STR2:= 'general/yAxisMin'),
			payload	:= '');	
	ELSE
		_Hmi.publish(
			topic	:= Tc2_Standard.CONCAT(STR1:= _topicPrefix, STR2:= 'general/yAxisMin'),
			payload	:= REAL_TO_STRING(_yMin));	
	END_IF
END_IF
(* Y Min Visible *)
IF (_yLastMinVisible <> _yMinVisible) OR _onHmiConnection.Q THEN
	_yLastMinVisible:= _yMinVisible;
	_yLastMin:= _yMin;
	IF NOT _yMinVisible THEN
		_Hmi.publish(
			topic	:= Tc2_Standard.CONCAT(STR1:= _topicPrefix, STR2:= 'general/yAxisMin'),
			payload	:= '');	
	ELSE
		_Hmi.publish(
			topic	:= Tc2_Standard.CONCAT(STR1:= _topicPrefix, STR2:= 'general/yAxisMin'),
			payload	:= REAL_TO_STRING(_yMin));	
	END_IF
END_IF
(* Y Max *)
IF ((_yLastMax <> _yMax) OR _onHmiConnection.Q) THEN
	_yLastMax:= _yMax;
	IF NOT _yMaxVisible THEN
		_Hmi.publish(
			topic	:= Tc2_Standard.CONCAT(STR1:= _topicPrefix, STR2:= 'general/yAxisMax'),
			payload	:= '');	
	ELSE
		_Hmi.publish(
			topic	:= Tc2_Standard.CONCAT(STR1:= _topicPrefix, STR2:= 'general/yAxisMax'),
			payload	:= REAL_TO_STRING(_yMax));		
	END_IF
END_IF
(* Y Max Visible *)
IF (_yLastMaxVisible <> _yMaxVisible) OR _onHmiConnection.Q THEN
	_yLastMaxVisible:= _yMaxVisible;
	_yLastMax:= _yMax;
	IF NOT _yMaxVisible THEN
		_Hmi.publish(
			topic	:= Tc2_Standard.CONCAT(STR1:= _topicPrefix, STR2:= 'general/yAxisMax'),
			payload	:= '');	
	ELSE
		_Hmi.publish(
			topic	:= Tc2_Standard.CONCAT(STR1:= _topicPrefix, STR2:= 'general/yAxisMax'),
			payload	:= REAL_TO_STRING(_yMax));		
	END_IF
END_IF
END_METHOD

METHOD FB_init : BOOL
VAR_INPUT
	bInitRetains	: BOOL; // if TRUE, the retain variables are initialized (warm start / cold start)
	bInCopyCode 	: BOOL;  // if TRUE, the instance afterwards gets moved into the copy code (online change)
	Hmi				: I_NexaHmi;
	id				: Tc2_System.T_MaxString;
	name			: Tc2_System.T_MaxString;
	xTitle			: STRING;
	yTitle			: STRING;
END_VAR
THIS^._Hmi:= Hmi;
THIS^._id:= id;
THIS^._name:= name;
THIS^._xTitle:= xTitle;
THIS^._yTitle:= yTitle;

FOR _counter:= 1 TO GVL_TcNexaHmiUtilities.numOfGraphLines2D DO
	_Lines[_counter].Hmi:= Hmi;
END_FOR
END_METHOD

PROPERTY description : Tc2_System.T_MaxString
GET
description:= _description;
END_GET
SET
_description:= description;
END_SET
END_PROPERTY

PROPERTY Lines : REFERENCE TO ARRAY[1..GVL_TcNexaHmiUtilities.numOfGraphLines2D] OF FB_NexaHmi_GraphLine2D
GET
Lines REF= _Lines;
END_GET
END_PROPERTY

PROPERTY PUBLIC xMax : REAL
GET
xMax:= _xMax;
END_GET
SET
_xMax:= xMax;
END_SET
END_PROPERTY

PROPERTY PUBLIC xMaxVisible : BOOL
GET
xMaxVisible:= _xMaxVisible;
END_GET
SET
_xMaxVisible:= xMaxVisible;
END_SET
END_PROPERTY

PROPERTY PUBLIC xMin : REAL
GET
xMin:= _xMin;
END_GET
SET
_xMin:= xMin;
END_SET
END_PROPERTY

PROPERTY PUBLIC xMinVisible : BOOL
GET
xMinVisible:= _xMinVisible;
END_GET
SET
_xMaxVisible:= xMaxVisible;
END_SET
END_PROPERTY

PROPERTY PUBLIC yMax : REAL
GET
yMax:= _yMax;
END_GET
SET
_yMax:= yMax;
END_SET
END_PROPERTY

PROPERTY PUBLIC yMaxVisible : BOOL
GET
yMaxVisible:= _yMaxVisible;
END_GET
SET
_yMaxVisible:= yMaxVisible;
END_SET
END_PROPERTY

PROPERTY PUBLIC yMin : REAL
GET
yMin:= _Ymin;
END_GET
SET
_yMin:= yMin;
END_SET
END_PROPERTY

PROPERTY PUBLIC yMinVisible : BOOL
GET
yMinVisible:= _yMinVisible;
END_GET
SET
_yMinVisible:= yMinVisible;
END_SET
END_PROPERTY

METHOD PUBLIC clear
VAR_INPUT
END_VAR
FOR _counter:= 1 TO GVL_TcNexaHmiUtilities.numOfGraphLines2D DO
	_Lines[_counter].clear();
END_FOR

_xMax:= 0;
_xMaxVisible:= FALSE;
_xMin:= 0;
_yMinVisible:= FALSE;
_yMax:= 0;
_yMaxVisible:= FALSE;
_yMin:= 0;
_yMinVisible:= FALSE;
END_METHOD

METHOD PUBLIC FB_main
VAR_INPUT
END_VAR
_isHmiConnected:= _Hmi.isConnected;
_onHmiConnection(CLK:= _isHmiConnected);

_onConnection();
_updateTopics();

FOR _counter:= 1 TO GVL_TcNexaHmiUtilities.numOfGraphLines2D DO
	_Lines[_counter].FB_main();
END_FOR
END_METHOD

METHOD PUBLIC publish
VAR_INPUT
END_VAR
FOR _counter:= 1 TO GVL_TcNexaHmiUtilities.numOfGraphLines2D DO
	_Lines[_counter].publish();
END_FOR
END_METHOD

END_FUNCTION_BLOCK

// Elements/Graph 2D/FB_NexaHmi_GraphLine2D
FUNCTION_BLOCK INTERNAL FB_NexaHmi_GraphLine2D
VAR
	_Hmi				: I_NexaHmi;
	_onHmiConnection	: Tc2_Standard.R_TRIG;
	_isHmiConnected		: BOOL;
	_topicPrefix		: Tc2_System.T_MaxString;
	_id					: Tc2_System.T_MaxString;
	_color				: E_GraphLineColor2D;
	_lastColor			: E_GraphLineColor2D;
	_buffer				: ARRAY[0..BUFFER_SIZE] OF BYTE;//STRING(BUFFER_SIZE);
	_bufferSize			: UDINT;
	_lastBufferSize		: UDINT;
	_timerUpdatePoints	: Tc2_Standard.TON;
	_FormatString		: Tc2_Utilities.FB_FormatString;
	_formattedString	: Tc2_System.T_MaxString;
	_stringLength		: UDINT;
	_tempX				: REAL;
	_tempY				: REAL;
END_VAR
VAR CONSTANT
	BUFFER_SIZE			: UDINT:= 10000;
END_VAR

METHOD PROTECTED _clearBuffer
VAR_INPUT
END_VAR
Tc2_System.MEMSET(
	destAddr	:= ADR(_buffer),
	fillByte	:= 0,
	n			:= SIZEOF(_buffer));
_bufferSize:= 0;
END_METHOD

METHOD PROTECTED _getColor : STRING
VAR_INPUT
END_VAR
IF (_color = E_GraphLineColor2D.black) THEN
	_getColor:= 'black';
ELSIF (_color = E_GraphLineColor2D.blue) THEN
	_getColor:= 'blue';
ELSIF (_color = E_GraphLineColor2D.green) THEN
	_getColor:= 'green';
ELSIF (_color = E_GraphLineColor2D.grey) THEN
	_getColor:= 'grey';
ELSIF (_color = E_GraphLineColor2D.purple) THEN
	_getColor:= 'purple';
ELSIF (_color = E_GraphLineColor2D.red) THEN
	_getColor:= 'red';
ELSIF (_color = E_GraphLineColor2D.yellow) THEN
	_getColor:= 'yellow';
END_IF
END_METHOD

METHOD PROTECTED _onConnection
VAR_INPUT
END_VAR
IF NOT _onHmiConnection.Q THEN RETURN; END_IF

_Hmi.publish(
	topic	:= Tc2_Standard.CONCAT(STR1:= _topicPrefix, STR2:= 'active'),
	payload	:= BOOL_TO_STRING(TRUE));
END_METHOD

METHOD PROTECTED _updateTopics
VAR_INPUT
END_VAR
IF NOT _isHmiConnected THEN RETURN; END_IF

(* Color *)
IF (_lastColor <> _color) OR _onHmiConnection.Q THEN
	_lastColor:= _color;
	_Hmi.publish(
		topic	:= Tc2_Standard.CONCAT(STR1:= _topicPrefix, STR2:= 'color'),
		payload	:= _getColor());
END_IF
//(* Points *)
//_timerUpdatePoints(IN:= _lastBufferSize <> _bufferSize, PT:= T#250MS);
//IF _timerUpdatePoints.Q THEN
//	_lastBufferSize:= _bufferSize;
//	_Hmi.publishAdr(
//		topic		:= Tc2_Standard.CONCAT(STR1:= _topicPrefix, STR2:= 'points'),
//		payload		:= ADR(_buffer),
//		payloadSize	:= _bufferSize);
//END_IF
END_METHOD

PROPERTY INTERNAL Hmi : I_NexaHmi
GET
Hmi:= _Hmi;
END_GET
SET
_Hmi:= Hmi;
END_SET
END_PROPERTY

PROPERTY INTERNAL topicPrefix : Tc2_System.T_MaxString
GET
topicPrefix:= _topicPrefix;
END_GET
SET
_topicPrefix:= topicPrefix;
END_SET
END_PROPERTY

METHOD PUBLIC addPoint
VAR_INPUT
	x	: REAL;
	y	: REAL;
END_VAR
_tempX:= x;
_tempY:= y;

_FormatString(
	sFormat	:= '%.2f,%.2f;',
	arg1	:= Tc2_Utilities.F_REAL(in:= _tempX),
	arg2	:= Tc2_Utilities.F_REAL(in:= _tempY),
	
	sOut	=> _formattedString);

_stringLength:= INT_TO_UDINT(Tc2_Standard.LEN(STR:= _formattedString));

IF ((_bufferSize + _stringLength) < BUFFER_SIZE) THEN
	Tc2_System.MEMCPY(
		destAddr	:= ADR(_buffer) + _bufferSize,
		srcAddr		:= ADR(_formattedString),
		n			:= _stringLength);
	
	_bufferSize:= _bufferSize + _stringLength;
END_IF






//_tempBufferSize:= _bufferSize + _stringLength;
//_tempBuffer:= __NEW(BYTE, _tempBufferSize);

//IF (_buffer <> 0) AND (_bufferSize > 0) THEN
//	Tc2_System.MEMCPY(
//		destAddr	:= _tempBuffer,
//		srcAddr		:= _buffer,
//		n			:= _bufferSize);
//	IF (_buffer <> 0) THEN __DELETE(_buffer); END_IF
//END_IF

//Tc2_System.MEMCPY(
//	destAddr	:= _tempBuffer + _bufferSize,
//	srcAddr		:= ADR(_formattedString),
//	n			:= _stringLength);
	
//_buffer:= _tempBuffer;
//_bufferSize:= _tempBufferSize;
END_METHOD

METHOD PUBLIC clear
VAR_INPUT
END_VAR
_clearBuffer();
END_METHOD

METHOD INTERNAL FB_main
VAR_INPUT
END_VAR
_isHmiConnected:= _Hmi.isConnected;
_onHmiConnection(CLK:= _isHmiConnected);

_onConnection();
_updateTopics();
END_METHOD

METHOD PUBLIC publish
VAR_INPUT
END_VAR
_Hmi.publishAdr(
	topic		:= Tc2_Standard.CONCAT(STR1:= _topicPrefix, STR2:= 'points'),
	payload		:= ADR(_buffer),
	payloadSize	:= _bufferSize);
END_METHOD

METHOD PUBLIC setColor
VAR_INPUT
	color		: E_GraphLineColor2D;
END_VAR
_color:= color;
END_METHOD

END_FUNCTION_BLOCK

// Elements/POUs/FB_CustomHmiButton
FUNCTION_BLOCK FB_CustomHmiButton
VAR
	_name		: STRING;
	_visible	: BOOL;
	_focused	: BOOL;
	_onTap		: BOOL;
END_VAR

PROPERTY focused : BOOL
GET
focused:= _focused;
END_GET
SET
_focused:= focused;
END_SET
END_PROPERTY

PROPERTY PUBLIC name : STRING
GET
name:= _name;
END_GET
SET
_name:= name;
END_SET
END_PROPERTY

PROPERTY PUBLIC onTap : BOOL
GET
onTap:= _onTap;
END_GET
SET
_onTap:= onTap;
END_SET
END_PROPERTY

PROPERTY PUBLIC visible : BOOL
GET
visible:= _visible;
END_GET
SET
_visible:= visible;
END_SET
END_PROPERTY

METHOD PUBLIC clear
VAR_INPUT
END_VAR
_name:= '';
_visible:= FALSE;
END_METHOD

END_FUNCTION_BLOCK

// Elements/POUs/FB_ModeHmiButton
FUNCTION_BLOCK FB_ModeHmiButton
VAR
	_enabled		: BOOL;
	_visible		: BOOL:= TRUE;
	_onTap			: BOOL;
	_onLongPress	: BOOL;
END_VAR

PROPERTY PUBLIC enabled : BOOL
GET
enabled:= _enabled;
END_GET
SET
_enabled:= enabled;
END_SET
END_PROPERTY

PROPERTY PUBLIC onLongPress : BOOL
GET
onLongPress:= _onLongPress;
END_GET
SET
_onLongPress:= onLongPress;
END_SET
END_PROPERTY

PROPERTY PUBLIC onTap : BOOL
GET
onTap:= _onTap;
END_GET
SET
_onTap:= onTap;
END_SET
END_PROPERTY

PROPERTY PUBLIC visible : BOOL
GET
visible:= _visible;
END_GET
SET
_visible:= visible;
END_SET
END_PROPERTY

METHOD PUBLIC clear
VAR_INPUT
END_VAR
_enabled:= FALSE;
_visible:= TRUE;
END_METHOD

METHOD clearCommand
VAR_INPUT
END_VAR
_onTap:= FALSE;
_onLongPress:= FALSE;
END_METHOD

END_FUNCTION_BLOCK

// Elements/POUs/FB_NexaHmiCustomButtons
FUNCTION_BLOCK FB_NexaHmiCustomButtons
VAR
	_Buttons			: ARRAY[1..GVL_TcNexaHmiUtilities.numOfCustomButtons] OF FB_CustomHmiButton;
END_VAR

PROPERTY PUBLIC Buttons : REFERENCE TO ARRAY[1..GVL_TcNexaHmiUtilities.numOfCustomButtons] OF FB_CustomHmiButton
GET
Buttons REF= _Buttons;
END_GET
END_PROPERTY

METHOD PUBLIC clear
VAR_INPUT
END_VAR
VAR
	_tmpCounter			: USINT;
END_VAR
FOR _tmpCounter:= 1 TO GVL_TcNexaHmiUtilities.numOfCustomButtons DO
	_Buttons[_tmpCounter].clear();
END_FOR
END_METHOD

END_FUNCTION_BLOCK

// Elements/POUs/FB_NexaHmiTextFields
FUNCTION_BLOCK FB_NexaHmiTextFields
VAR
	_fields			: ARRAY[1..GVL_TcNexaHmiUtilities.numOfTextFields] OF Tc2_System.T_MaxString;
	_userAction		: BOOL;
END_VAR

PROPERTY PUBLIC fields : REFERENCE TO ARRAY[1..GVL_TcNexaHmiUtilities.numOfTextFields] OF Tc2_System.T_MaxString
GET
fields REF= _fields;
END_GET
END_PROPERTY

PROPERTY PUBLIC userAction : BOOL
GET
userAction:= _userAction;
END_GET
SET
_userAction:= userAction;
END_SET
END_PROPERTY

METHOD PUBLIC clear
VAR
	_tmpCounter		: USINT;	
END_VAR
FOR _tmpCounter:= 1 TO GVL_TcNexaHmiUtilities.numOfTextFields DO
	_fields[_tmpCounter]:= '';
END_FOR
_userAction:= FALSE;
END_METHOD

END_FUNCTION_BLOCK

// Order/FB_NexaHmiOrderBOOL
FUNCTION_BLOCK FB_NexaHmiOrderBOOL
VAR
	_Hmi				: I_NexaHmi;
	_onHmiConnection	: Tc2_Standard.R_TRIG;
	_isHmiConnected		: BOOL;
	_id					: UINT;
	_cellTag			: STRING;
	_name				: Tc2_System.T_MaxString;
	_description		: Tc2_System.T_MaxString;
	_value				: BOOL;
	_defaultValue		: BOOL;
	_enabled			: BOOL;
	(* General *)
	_timerPublish		: Tc2_Standard.TON;
	_topicPrefix		: Tc2_System.T_MaxString;
	(* Last values *)
	_lastValue			: BOOL;
	_lastEnabled		: BOOL;
END_VAR

METHOD PROTECTED _handleNewMessages
VAR_INPUT
END_VAR
IF NOT _isHmiConnected THEN RETURN; END_IF

IF _Hmi.onNewMessage THEN
	IF (Tc2_Standard.FIND(STR1:= _Hmi.messageFullTopic, STR2:= _topicPrefix) <> 0) THEN
		IF (_Hmi.messageFullTopic = Tc2_Standard.CONCAT(STR1:= _topicPrefix, STR2:= 'value')) THEN
			_value:= STRING_TO_BOOL(_Hmi.messagePayload);
			_lastValue:= _value;
		END_IF
	END_IF
END_IF
END_METHOD

METHOD PROTECTED _onConnection
VAR_INPUT
END_VAR
IF NOT _onHmiConnection.Q THEN RETURN; END_IF

_topicPrefix:= Tc2_Standard.CONCAT(STR1:= _cellTag, STR2:= '/order/settings/booleans/');
_topicPrefix:= Tc2_Standard.CONCAT(STR1:= _topicPrefix, STR2:= UINT_TO_STRING(_id));
_topicPrefix:= Tc2_Standard.CONCAT(STR1:= _topicPrefix, STR2:= '/');
_Hmi.subscribe(topic:= Tc2_Standard.CONCAT(STR1:= _topicPrefix, STR2:= 'value'));

_Hmi.publish(
	topic	:= Tc2_Standard.CONCAT(STR1:= _topicPrefix, STR2:= 'active'),
	payload	:= BOOL_TO_STRING(TRUE));
_Hmi.publish(
	topic	:= Tc2_Standard.CONCAT(STR1:= _topicPrefix, STR2:= 'name'),
	payload	:= _name);
_Hmi.publish(
	topic	:= Tc2_Standard.CONCAT(STR1:= _topicPrefix, STR2:= 'description'),
	payload	:= _description);
END_METHOD

METHOD PROTECTED _updateTopics
VAR_INPUT
END_VAR
IF NOT _isHmiConnected THEN RETURN; END_IF

(* Value *)
IF (_lastValue <> _value) AND _timerPublish.Q THEN
	_lastValue:= _value;
	_Hmi.publish(
		topic	:= Tc2_Standard.CONCAT(STR1:= _topicPrefix, STR2:= 'value'),
		payload	:= BOOL_TO_STRING(_value));
END_IF
(* Enabled *)
IF (_lastEnabled <> _enabled) OR _onHmiConnection.Q THEN
	_lastEnabled:= _enabled;
	_Hmi.publish(
		topic	:= Tc2_Standard.CONCAT(STR1:= _topicPrefix, STR2:= 'enabled'),
		payload	:= BOOL_TO_STRING(_enabled));
END_IF
END_METHOD

METHOD FB_init : BOOL
VAR_INPUT
	bInitRetains	: BOOL; // if TRUE, the retain variables are initialized (warm start / cold start)
	bInCopyCode 	: BOOL;  // if TRUE, the instance afterwards gets moved into the copy code (online change)
	Hmi				: I_NexaHmi;
	cellTag			: STRING;
	id				: UINT;
	name			: Tc2_System.T_MaxString;
	description		: Tc2_System.T_MaxString;
	defaultValue	: BOOL;
END_VAR
THIS^._Hmi:= Hmi;
THIS^._id:= id;
THIS^._name:= name;
THIS^._description:= description;
THIS^._defaultValue:= defaultValue;
THIS^._value:= defaultValue;
THIS^._cellTag:= cellTag;
END_METHOD

PROPERTY description : Tc2_System.T_MaxString
GET
description:= _description;
END_GET
END_PROPERTY

PROPERTY name : Tc2_System.T_MaxString
GET
name:= _name;
END_GET
END_PROPERTY

PROPERTY PUBLIC value : BOOL
GET
value:= _value;
END_GET
SET
_value:= value;
END_SET
END_PROPERTY

METHOD PUBLIC FB_main
VAR_INPUT
END_VAR
_timerPublish(IN:= _isHmiConnected, PT:= T#1S);
_isHmiConnected:= _Hmi.isConnected;
_onHmiConnection(CLK:= _isHmiConnected);

_onConnection();
_updateTopics();
_handleNewMessages();
END_METHOD

END_FUNCTION_BLOCK

// Order/FB_NexaHmiOrderINT
FUNCTION_BLOCK FB_NexaHmiOrderINT
VAR
	_Hmi				: I_NexaHmi;
	_onHmiConnection	: Tc2_Standard.R_TRIG;
	_isHmiConnected		: BOOL;
	_id					: UINT;
	_cellTag			: STRING;
	_name				: Tc2_System.T_MaxString;
	_description		: Tc2_System.T_MaxString;
	_value				: INT;
	_defaultValue		: INT;
	_lowerLimit			: INT:= -32768;
	_hasLowerLimit		: BOOL;
	_upperLimit			: INT:= 32767;
	_hasUpperLimit		: BOOL;
	_unit				: STRING;
	_enabled			: BOOL;
	(* General *)
	_timerPublish		: Tc2_Standard.TON;
	_topicPrefix		: Tc2_System.T_MaxString;
	(* Last values *)
	_lastValue			: INT;
	_lastEnabled		: BOOL;
END_VAR

METHOD PROTECTED _handleNewMessage
VAR_INPUT
END_VAR
IF NOT _isHmiConnected THEN RETURN; END_IF

IF _Hmi.onNewMessage THEN
	IF (Tc2_Standard.FIND(STR1:= _Hmi.messageFullTopic, STR2:= _topicPrefix) <> 0) THEN
		IF (_Hmi.messageFullTopic = Tc2_Standard.CONCAT(STR1:= _topicPrefix, STR2:= 'value')) THEN
			_value:= STRING_TO_INT(_Hmi.messagePayload);
			_lastValue:= _value;
		END_IF
	END_IF
END_IF
END_METHOD

METHOD PROTECTED _onConnection
VAR_INPUT
END_VAR
IF NOT _onHmiConnection.Q THEN RETURN; END_IF

_topicPrefix:= Tc2_Standard.CONCAT(STR1:= _cellTag, STR2:= '/order/settings/integers/');
_topicPrefix:= Tc2_Standard.CONCAT(STR1:= _topicPrefix, STR2:= UINT_TO_STRING(_id));
_topicPrefix:= Tc2_Standard.CONCAT(STR1:= _topicPrefix, STR2:= '/');
_Hmi.subscribe(topic:= Tc2_Standard.CONCAT(STR1:= _topicPrefix, STR2:= 'value'));

_Hmi.publish(
	topic	:= Tc2_Standard.CONCAT(STR1:= _topicPrefix, STR2:= 'active'),
	payload	:= BOOL_TO_STRING(TRUE));
_Hmi.publish(
	topic	:= Tc2_Standard.CONCAT(STR1:= _topicPrefix, STR2:= 'name'),
	payload	:= _name);
_Hmi.publish(
	topic	:= Tc2_Standard.CONCAT(STR1:= _topicPrefix, STR2:= 'description'),
	payload	:= _description);
_Hmi.publish(
	topic	:= Tc2_Standard.CONCAT(STR1:= _topicPrefix, STR2:= 'unit'),
	payload	:= _unit);
(* Upper Value *)
IF _hasLowerLimit THEN
	_Hmi.publish(
		topic	:= Tc2_Standard.CONCAT(STR1:= _topicPrefix, STR2:= 'min'),
		payload	:= INT_TO_STRING(_lowerLimit));
END_IF
IF _hasUpperLimit THEN
	_Hmi.publish(
		topic	:= Tc2_Standard.CONCAT(STR1:= _topicPrefix, STR2:= 'max'),
		payload	:= INT_TO_STRING(_upperLimit));
END_IF
END_METHOD

METHOD PROTECTED _updateTopics
VAR_INPUT
END_VAR
IF NOT _isHmiConnected THEN RETURN; END_IF

(* Value *)
IF (_lastValue <> _value) AND _timerPublish.Q THEN
	_lastValue:= _value;
	_Hmi.publish(
		topic	:= Tc2_Standard.CONCAT(STR1:= _topicPrefix, STR2:= 'value'),
		payload	:= INT_TO_STRING(_value));
END_IF
END_METHOD

METHOD FB_init : BOOL
VAR_INPUT
	bInitRetains	: BOOL; // if TRUE, the retain variables are initialized (warm start / cold start)
	bInCopyCode 	: BOOL;  // if TRUE, the instance afterwards gets moved into the copy code (online change)
	Hmi				: I_NexaHmi;
	cellTag			: STRING;
	id				: UINT;
	name			: Tc2_System.T_MaxString;
	description		: Tc2_System.T_MaxString;
	defaultValue	: INT;
	lowerLimit		: INT;
	hasLowerLimit	: BOOL;
	upperLimit		: INT;
	hasUpperLimit	: BOOL;
	unit			: STRING;
END_VAR
THIS^._Hmi:= Hmi;
THIS^._id:= id;
THIS^._name:= name;
THIS^._description:= description;
THIS^._defaultValue:= defaultValue;
THIS^._value:= defaultValue;
THIS^._lowerLimit:= lowerLimit;
THIS^._hasLowerLimit:= hasLowerLimit;
THIS^._upperLimit:= upperLimit;
THIS^._hasUpperLimit:= hasUpperLimit;
THIS^._unit:= unit;
THIS^._cellTag:= cellTag;
END_METHOD

PROPERTY description : Tc2_System.T_MaxString
GET
description:= _description;
END_GET
END_PROPERTY

PROPERTY PUBLIC lowerLimit : INT
GET
lowerLimit:= _lowerLimit;
END_GET
END_PROPERTY

PROPERTY name : Tc2_System.T_MaxString
GET
name:= _name;
END_GET
END_PROPERTY

PROPERTY PUBLIC upperLimit : INT
GET
upperLimit:= _upperLimit;
END_GET
END_PROPERTY

PROPERTY PUBLIC value : INT
GET
value:= _value;
END_GET
SET
_value:= value;
END_SET
END_PROPERTY

METHOD PUBLIC FB_main
VAR_INPUT
END_VAR
_timerPublish(IN:= _isHmiConnected, PT:= T#1S);
_isHmiConnected:= _Hmi.isConnected;
_onHmiConnection(CLK:= _isHmiConnected);

_onConnection();
_updateTopics();
_handleNewMessage();
END_METHOD

END_FUNCTION_BLOCK

// Order/FB_NexaHmiOrderREAL
FUNCTION_BLOCK FB_NexaHmiOrderREAL
VAR
	_Hmi				: I_NexaHmi;
	_onHmiConnection	: Tc2_Standard.R_TRIG;
	_isHmiConnected		: BOOL;
	_id					: UINT;
	_cellTag			: STRING;
	_name				: Tc2_System.T_MaxString;
	_description		: Tc2_System.T_MaxString;
	_value				: REAL;
	_defaultValue		: REAL;
	_lowerLimit			: REAL:= -3.402823E+38;
	_hasLowerLimit		: BOOL;
	_upperLimit			: REAL:= 3.402823E+38;
	_hasUpperLimit		: BOOL;
	_unit				: STRING;
	(* General *)
	_timerPublish		: Tc2_Standard.TON;
	_topicPrefix		: Tc2_System.T_MaxString;
	(* Last values *)
	_lastValue			: REAL;
END_VAR

METHOD PROTECTED _handleNewMessage
VAR_INPUT
END_VAR
IF NOT _isHmiConnected THEN RETURN; END_IF

IF _Hmi.onNewMessage THEN
	IF (Tc2_Standard.FIND(STR1:= _Hmi.messageFullTopic, STR2:= _topicPrefix) <> 0) THEN
		IF (_Hmi.messageFullTopic = Tc2_Standard.CONCAT(STR1:= _topicPrefix, STR2:= 'value')) THEN
			_value:= STRING_TO_REAL(_Hmi.messagePayload);
			_lastValue:= _value;
		END_IF
	END_IF
END_IF
END_METHOD

METHOD PROTECTED _onConnection
VAR_INPUT
END_VAR
IF NOT _onHmiConnection.Q THEN RETURN; END_IF

_topicPrefix:= Tc2_Standard.CONCAT(STR1:= _cellTag, STR2:= '/order/settings/reals/');
_topicPrefix:= Tc2_Standard.CONCAT(STR1:= _topicPrefix, STR2:= UINT_TO_STRING(_id));
_topicPrefix:= Tc2_Standard.CONCAT(STR1:= _topicPrefix, STR2:= '/');
_Hmi.subscribe(topic:= Tc2_Standard.CONCAT(STR1:= _topicPrefix, STR2:= 'value'));

_Hmi.publish(
	topic	:= Tc2_Standard.CONCAT(STR1:= _topicPrefix, STR2:= 'active'),
	payload	:= BOOL_TO_STRING(TRUE));
_Hmi.publish(
	topic	:= Tc2_Standard.CONCAT(STR1:= _topicPrefix, STR2:= 'name'),
	payload	:= _name);
_Hmi.publish(
	topic	:= Tc2_Standard.CONCAT(STR1:= _topicPrefix, STR2:= 'description'),
	payload	:= _description);
_Hmi.publish(
	topic	:= Tc2_Standard.CONCAT(STR1:= _topicPrefix, STR2:= 'unit'),
	payload	:= _unit);
(* Upper Value *)
IF _hasLowerLimit THEN
	_Hmi.publish(
		topic	:= Tc2_Standard.CONCAT(STR1:= _topicPrefix, STR2:= 'min'),
		payload	:= REAL_TO_STRING(_lowerLimit));
END_IF
IF _hasUpperLimit THEN
	_Hmi.publish(
		topic	:= Tc2_Standard.CONCAT(STR1:= _topicPrefix, STR2:= 'max'),
		payload	:= REAL_TO_STRING(_upperLimit));
END_IF
END_METHOD

METHOD PROTECTED _updateTopics
VAR_INPUT
END_VAR
IF NOT _isHmiConnected THEN RETURN; END_IF

(* Value *)
IF (_lastValue <> _value) AND _timerPublish.Q THEN
	_lastValue:= _value;
	_Hmi.publish(
		topic	:= Tc2_Standard.CONCAT(STR1:= _topicPrefix, STR2:= 'value'),
		payload	:= REAL_TO_STRING(_value));
END_IF
END_METHOD

METHOD FB_init : BOOL
VAR_INPUT
	bInitRetains	: BOOL; // if TRUE, the retain variables are initialized (warm start / cold start)
	bInCopyCode 	: BOOL;  // if TRUE, the instance afterwards gets moved into the copy code (online change)
	Hmi				: I_NexaHmi;
	cellTag			: STRING;
	id				: UINT;
	name			: Tc2_System.T_MaxString;
	description		: Tc2_System.T_MaxString;
	defaultValue	: REAL;
	lowerLimit		: REAL;
	hasLowerLimit	: BOOL;
	upperLimit		: REAL;
	hasUpperLimit	: BOOL;
	unit			: STRING;
END_VAR
THIS^._Hmi:= Hmi;
THIS^._id:= id;
THIS^._name:= name;
THIS^._description:= description;
THIS^._defaultValue:= defaultValue;
THIS^._value:= defaultValue;
THIS^._lowerLimit:= lowerLimit;
THIS^._hasLowerLimit:= hasLowerLimit;
THIS^._upperLimit:= upperLimit;
THIS^._hasUpperLimit:= hasUpperLimit;
THIS^._unit:= unit;
THIS^._cellTag:= cellTag;
END_METHOD

PROPERTY description : Tc2_System.T_MaxString
GET
description:= _description;
END_GET
END_PROPERTY

PROPERTY PUBLIC lowerLimit : REAL
GET
lowerLimit:= _lowerLimit;
END_GET
END_PROPERTY

PROPERTY name : Tc2_System.T_MaxString
GET
name:= _name;
END_GET
END_PROPERTY

PROPERTY PUBLIC upperLimit : REAL
GET
upperLimit:= _upperLimit;
END_GET
END_PROPERTY

PROPERTY PUBLIC value : REAL
GET
value:= _value;
END_GET
SET
_value:= value;
END_SET
END_PROPERTY

METHOD PUBLIC FB_main
VAR_INPUT
END_VAR
_timerPublish(IN:= _isHmiConnected, PT:= T#1S);
_isHmiConnected:= _Hmi.isConnected;
_onHmiConnection(CLK:= _isHmiConnected);

_onConnection();
_updateTopics();
_handleNewMessage();
END_METHOD

END_FUNCTION_BLOCK

// Order/FB_NexaHmiOrderSTRING
FUNCTION_BLOCK FB_NexaHmiOrderSTRING
VAR
	_Hmi				: I_NexaHmi;
	_onHmiConnection	: Tc2_Standard.R_TRIG;
	_isHmiConnected		: BOOL;
	_id					: UINT;
	_cellTag			: STRING;
	_name				: Tc2_System.T_MaxString;
	_description		: Tc2_System.T_MaxString;
	_value				: Tc2_System.T_MaxString;
	_defaultValue		: Tc2_System.T_MaxString;
	(* General *)
	_timerPublish		: Tc2_Standard.TON;
	_topicPrefix		: Tc2_System.T_MaxString;
	(* Last values *)
	_lastValue			: Tc2_System.T_MaxString;
END_VAR

METHOD PROTECTED _handleNewMessages
VAR_INPUT
END_VAR
IF NOT _isHmiConnected THEN RETURN; END_IF

IF _Hmi.onNewMessage THEN
	IF (Tc2_Standard.FIND(STR1:= _Hmi.messageFullTopic, STR2:= _topicPrefix) <> 0) THEN
		IF (_Hmi.messageFullTopic = Tc2_Standard.CONCAT(STR1:= _topicPrefix, STR2:= 'value')) THEN
			_value:= _Hmi.messagePayload;
			_lastValue:= _value;
		END_IF
	END_IF
END_IF
END_METHOD

METHOD PROTECTED _onConnection
VAR_INPUT
END_VAR
IF NOT _onHmiConnection.Q THEN RETURN; END_IF

_topicPrefix:= Tc2_Standard.CONCAT(STR1:= _cellTag, STR2:= '/order/settings/strings/');
_topicPrefix:= Tc2_Standard.CONCAT(STR1:= _topicPrefix, STR2:= UINT_TO_STRING(_id));
_topicPrefix:= Tc2_Standard.CONCAT(STR1:= _topicPrefix, STR2:= '/');
_Hmi.subscribe(topic:= Tc2_Standard.CONCAT(STR1:= _topicPrefix, STR2:= 'value'));

_Hmi.publish(
	topic	:= Tc2_Standard.CONCAT(STR1:= _topicPrefix, STR2:= 'active'),
	payload	:= BOOL_TO_STRING(TRUE));
_Hmi.publish(
	topic	:= Tc2_Standard.CONCAT(STR1:= _topicPrefix, STR2:= 'name'),
	payload	:= _name);
_Hmi.publish(
	topic	:= Tc2_Standard.CONCAT(STR1:= _topicPrefix, STR2:= 'description'),
	payload	:= _description);
END_METHOD

METHOD PROTECTED _updateTopics
VAR_INPUT
END_VAR
IF NOT _isHmiConnected THEN RETURN; END_IF

(* Value *)
IF (_lastValue <> _value) AND _timerPublish.Q THEN
	_lastValue:= _value;
	_Hmi.publish(
		topic	:= Tc2_Standard.CONCAT(STR1:= _topicPrefix, STR2:= 'value'),
		payload	:= _value);
END_IF
END_METHOD

METHOD FB_init : BOOL
VAR_INPUT
	bInitRetains	: BOOL; // if TRUE, the retain variables are initialized (warm start / cold start)
	bInCopyCode 	: BOOL;  // if TRUE, the instance afterwards gets moved into the copy code (online change)
	Hmi				: I_NexaHmi;
	cellTag			: STRING;
	id				: UINT;
	name			: Tc2_System.T_MaxString;
	description		: Tc2_System.T_MaxString;
	defaultValue	: Tc2_System.T_MaxString;
END_VAR
THIS^._Hmi:= Hmi;
THIS^._id:= id;
THIS^._name:= name;
THIS^._defaultValue:= defaultValue;
THIS^._value:= defaultValue;
THIS^._cellTag:= cellTag;
END_METHOD

PROPERTY PUBLIC value : STRING
GET
value:= _value;
END_GET
SET
_value:= value;
END_SET
END_PROPERTY

METHOD PUBLIC FB_main
VAR_INPUT
END_VAR
_timerPublish(IN:= _isHmiConnected, PT:= T#1S);
_isHmiConnected:= _Hmi.isConnected;
_onHmiConnection(CLK:= _isHmiConnected);

_onConnection();
_updateTopics();
_handleNewMessages();
END_METHOD

END_FUNCTION_BLOCK

// Order/FB_NexaHmiOrderTIME
FUNCTION_BLOCK FB_NexaHmiOrderTIME
VAR
	_Hmi				: I_NexaHmi;
	_onHmiConnection	: Tc2_Standard.R_TRIG;
	_isHmiConnected		: BOOL;
	_id					: UINT;
	_cellTag			: STRING;
	_name				: Tc2_System.T_MaxString;
	_description		: Tc2_System.T_MaxString;
	_value				: TIME;
	_defaultValue		: TIME;
	_lowerLimit			: TIME;
	_hasLowerLimit		: BOOL;
	_upperLimit			: TIME;
	_hasUpperLimit		: BOOL;
	(* General *)
	_timerPublish		: Tc2_Standard.TON;
	_topicPrefix		: Tc2_System.T_MaxString;
	(* Last values *)
	_lastValue			: TIME;
END_VAR

METHOD PROTECTED _handleNewMessages
VAR_INPUT
END_VAR
IF NOT _isHmiConnected THEN RETURN; END_IF

IF _Hmi.onNewMessage THEN
	IF (Tc2_Standard.FIND(STR1:= _Hmi.messageFullTopic, STR2:= _topicPrefix) <> 0) THEN
		IF (_Hmi.messageFullTopic = Tc2_Standard.CONCAT(STR1:= _topicPrefix, STR2:= 'value')) THEN
			_value:= UDINT_TO_TIME(STRING_TO_UDINT(_Hmi.messagePayload));
			_lastValue:= _value;
		END_IF
	END_IF
END_IF
END_METHOD

METHOD PROTECTED _onConnection
VAR_INPUT
END_VAR
IF NOT _onHmiConnection.Q THEN RETURN; END_IF

_topicPrefix:= Tc2_Standard.CONCAT(STR1:= _cellTag, STR2:= '/order/settings/times/');
_topicPrefix:= Tc2_Standard.CONCAT(STR1:= _topicPrefix, STR2:= UINT_TO_STRING(_id));
_topicPrefix:= Tc2_Standard.CONCAT(STR1:= _topicPrefix, STR2:= '/');
_Hmi.subscribe(topic:= Tc2_Standard.CONCAT(STR1:= _topicPrefix, STR2:= 'value'));

_Hmi.publish(
	topic	:= Tc2_Standard.CONCAT(STR1:= _topicPrefix, STR2:= 'active'),
	payload	:= BOOL_TO_STRING(TRUE));
_Hmi.publish(
	topic	:= Tc2_Standard.CONCAT(STR1:= _topicPrefix, STR2:= 'name'),
	payload	:= _name);
_Hmi.publish(
	topic	:= Tc2_Standard.CONCAT(STR1:= _topicPrefix, STR2:= 'description'),
	payload	:= _description);
(* Upper Value *)
IF _hasLowerLimit THEN
	_Hmi.publish(
		topic	:= Tc2_Standard.CONCAT(STR1:= _topicPrefix, STR2:= 'min'),
		payload	:= UDINT_TO_STRING(TIME_TO_UDINT(_lowerLimit)));
END_IF
IF _hasUpperLimit THEN
	_Hmi.publish(
		topic	:= Tc2_Standard.CONCAT(STR1:= _topicPrefix, STR2:= 'max'),
		payload	:= UDINT_TO_STRING(TIME_TO_UDINT(_upperLimit)));
END_IF
END_METHOD

METHOD PROTECTED _updateTopics
VAR_INPUT
END_VAR
IF NOT _isHmiConnected THEN RETURN; END_IF

(* Value *)
IF (_lastValue <> _value) AND _timerPublish.Q THEN
	_lastValue:= _value;
	_Hmi.publish(
		topic	:= Tc2_Standard.CONCAT(STR1:= _topicPrefix, STR2:= 'value'),
		payload	:= UDINT_TO_STRING(TIME_TO_UDINT(_value)));
END_IF
END_METHOD

METHOD FB_init : BOOL
VAR_INPUT
	bInitRetains	: BOOL; // if TRUE, the retain variables are initialized (warm start / cold start)
	bInCopyCode 	: BOOL;  // if TRUE, the instance afterwards gets moved into the copy code (online change)
	Hmi				: I_NexaHmi;
	cellTag			: STRING;
	id				: UINT;
	name			: Tc2_System.T_MaxString;
	description		: Tc2_System.T_MaxString;
	defaultValue	: TIME;
	lowerLimit		: TIME;
	hasLowerLimit	: BOOL;
	upperLimit		: TIME;
	hasUpperLimit	: BOOL;
END_VAR
THIS^._Hmi:= Hmi;
THIS^._id:= id;
THIS^._name:= name;
THIS^._description:= description;
THIS^._defaultValue:= defaultValue;
THIS^._value:= defaultValue;
THIS^._lowerLimit:= lowerLimit;
THIS^._hasLowerLimit:= hasLowerLimit;
THIS^._upperLimit:= upperLimit;
THIS^._hasUpperLimit:= hasUpperLimit;
THIS^._cellTag:= cellTag;
END_METHOD

PROPERTY description : Tc2_System.T_MaxString
GET
description:= _description;
END_GET
END_PROPERTY

PROPERTY name : Tc2_System.T_MaxString
GET
name:= _name;
END_GET
SET
_name:= name;
END_SET
END_PROPERTY

PROPERTY PUBLIC value : TIME
GET
value:= _value;
END_GET
SET
_value:= value;
END_SET
END_PROPERTY

METHOD PUBLIC FB_main
VAR_INPUT
END_VAR
_timerPublish(IN:= _isHmiConnected, PT:= T#1S);
_isHmiConnected:= _Hmi.isConnected;
_onHmiConnection(CLK:= _isHmiConnected);

_onConnection();
_updateTopics();
_handleNewMessages();
END_METHOD

END_FUNCTION_BLOCK

// Persistent/FB_NexaHmiPersistentBase
FUNCTION_BLOCK ABSTRACT FB_NexaHmiPersistentBase
VAR
	_Hmi				: I_NexaHmi;
	_onHmiConnection	: Tc2_Standard.R_TRIG;
	_isHmiConnected		: BOOL;
	_id					: STRING(255);
	(* General *)
	_timerPublish		: Tc2_Standard.TON;
	_topicPrefix		: STRING(255);
END_VAR

METHOD PROTECTED ABSTRACT _handleVar
VAR_INPUT
END_VAR
END_METHOD

METHOD PROTECTED _onConnection
VAR_INPUT
END_VAR
IF NOT _onHmiConnection.Q THEN RETURN; END_IF

_topicPrefix:= Tc2_Standard.CONCAT(STR1:= _Hmi.topicPrefix, STR2:= 'persistent/');
_topicPrefix:= Tc2_Standard.CONCAT(STR1:= _topicPrefix, STR2:= _id);
_topicPrefix:= Tc2_Standard.CONCAT(STR1:= _topicPrefix, STR2:= '/');
_Hmi.subscribe(topic:= Tc2_Standard.CONCAT(STR1:= _topicPrefix, STR2:= 'value'));
END_METHOD

METHOD FB_init : BOOL
VAR_INPUT
	bInitRetains	: BOOL; 	// if TRUE, the retain variables are initialized (warm start / cold start)
	bInCopyCode 	: BOOL;  	// if TRUE, the instance afterwards gets moved into the copy code (online change)
	Hmi				: I_NexaHmi;
	id				: Tc2_System.T_MaxString;
END_VAR
THIS^._Hmi:= Hmi;
THIS^._id:= id;
END_METHOD

METHOD PUBLIC FB_main
VAR_INPUT
END_VAR
_timerPublish(IN:= _isHmiConnected, PT:= T#1S);
_isHmiConnected:= _Hmi.isConnected;
_onHmiConnection(CLK:= _isHmiConnected);

_onConnection();
_handleVar();
END_METHOD

END_FUNCTION_BLOCK

// Persistent/FB_NexaHmiPersistentBOOL
FUNCTION_BLOCK FB_NexaHmiPersistentBOOL EXTENDS FB_NexaHmiPersistentBase
VAR
	_value				: BOOL;
	(* Last values *)
	_lastValue			: BOOL;
END_VAR

METHOD PROTECTED _handleVar
VAR_INPUT
END_VAR
IF NOT _isHmiConnected THEN RETURN; END_IF

(* Handle new messages *)
IF _Hmi.onNewMessage THEN
	IF (Tc2_Standard.FIND(STR1:= _Hmi.messageFullTopic, STR2:= _topicPrefix) <> 0) THEN
		IF (_Hmi.messageFullTopic = Tc2_Standard.CONCAT(STR1:= _topicPrefix, STR2:= 'value')) THEN
			_value:= STRING_TO_BOOL(_Hmi.messagePayload);
			_lastValue:= _value;
		END_IF
	END_IF
END_IF

(* Publish new messages *)
(* Value *)
IF (_lastValue <> _value) AND _timerPublish.Q THEN
	_lastValue:= _value;
	_Hmi.publish(
		topic	:= Tc2_Standard.CONCAT(STR1:= _topicPrefix, STR2:= 'value'),
		payload	:= BOOL_TO_STRING(_value));
END_IF
END_METHOD

METHOD FB_init : BOOL
VAR_INPUT
	bInitRetains	: BOOL; 	// if TRUE, the retain variables are initialized (warm start / cold start)
	bInCopyCode 	: BOOL;  	// if TRUE, the instance afterwards gets moved into the copy code (online change)
	Hmi				: I_NexaHmi;
	id				: Tc2_System.T_MaxString;
	defaultValue	: BOOL;
END_VAR
THIS^._value:= defaultValue;
END_METHOD

PROPERTY PUBLIC value : BOOL
GET
value:= _value;
END_GET
SET
_value:= value;
END_SET
END_PROPERTY

END_FUNCTION_BLOCK

// Persistent/FB_NexaHmiPersistentINT
FUNCTION_BLOCK FB_NexaHmiPersistentINT EXTENDS FB_NexaHmiPersistentBase
VAR
	_value				: INT;
	(* Last values *)
	_lastValue			: INT;
END_VAR

METHOD PROTECTED _handleVar
VAR_INPUT
END_VAR
IF NOT _isHmiConnected THEN RETURN; END_IF

(* Handle new messages *)
IF _Hmi.onNewMessage THEN
	IF (Tc2_Standard.FIND(STR1:= _Hmi.messageFullTopic, STR2:= _topicPrefix) <> 0) THEN
		IF (_Hmi.messageFullTopic = Tc2_Standard.CONCAT(STR1:= _topicPrefix, STR2:= 'value')) THEN
			_value:= STRING_TO_INT(_Hmi.messagePayload);
			_lastValue:= _value;
		END_IF
	END_IF
END_IF

(* Publish new messages *)
(* Value *)
IF (_lastValue <> _value) AND _timerPublish.Q THEN
	_lastValue:= _value;
	_Hmi.publish(
		topic	:= Tc2_Standard.CONCAT(STR1:= _topicPrefix, STR2:= 'value'),
		payload	:= INT_TO_STRING(_value));
END_IF
END_METHOD

METHOD FB_init : BOOL
VAR_INPUT
	bInitRetains	: BOOL; // if TRUE, the retain variables are initialized (warm start / cold start)
	bInCopyCode 	: BOOL;  // if TRUE, the instance afterwards gets moved into the copy code (online change)
	Hmi				: I_NexaHmi;
	id				: Tc2_System.T_MaxString;
	defaultValue	: INT;
END_VAR
THIS^._value:= defaultValue;
END_METHOD

PROPERTY PUBLIC value : INT
GET
value:= _value;
END_GET
SET
_value:= value;
END_SET
END_PROPERTY

END_FUNCTION_BLOCK

// Persistent/FB_NexaHmiPersistentREAL
FUNCTION_BLOCK FB_NexaHmiPersistentREAL EXTENDS FB_NexaHmiPersistentBase
VAR
	_value				: REAL;
	(* Last values *)
	_lastValue			: REAL;
END_VAR

METHOD PROTECTED _handleVar
VAR_INPUT
END_VAR
IF NOT _isHmiConnected THEN RETURN; END_IF

(* Handle new messages *)
IF _Hmi.onNewMessage THEN
	IF (Tc2_Standard.FIND(STR1:= _Hmi.messageFullTopic, STR2:= _topicPrefix) <> 0) THEN
		IF (_Hmi.messageFullTopic = Tc2_Standard.CONCAT(STR1:= _topicPrefix, STR2:= 'value')) THEN
			_value:= STRING_TO_REAL(_Hmi.messagePayload);
			_lastValue:= _value;
		END_IF
	END_IF
END_IF

(* Publish new messages *)
(* Value *)
IF (_lastValue <> _value) AND _timerPublish.Q THEN
	_lastValue:= _value;
	_Hmi.publish(
		topic	:= Tc2_Standard.CONCAT(STR1:= _topicPrefix, STR2:= 'value'),
		payload	:= REAL_TO_STRING(_value));
END_IF
END_METHOD

METHOD FB_init : BOOL
VAR_INPUT
	bInitRetains	: BOOL; // if TRUE, the retain variables are initialized (warm start / cold start)
	bInCopyCode 	: BOOL;  // if TRUE, the instance afterwards gets moved into the copy code (online change)
	Hmi				: I_NexaHmi;
	id				: Tc2_System.T_MaxString;
	defaultValue	: REAL;
END_VAR
THIS^._value:= defaultValue;
END_METHOD

PROPERTY PUBLIC value : REAL
GET
value:= _value;
END_GET
SET
_value:= value;
END_SET
END_PROPERTY

END_FUNCTION_BLOCK

// Persistent/FB_NexaHmiPersistentSTRING
FUNCTION_BLOCK FB_NexaHmiPersistentSTRING EXTENDS FB_NexaHmiPersistentBase
VAR
	_value				: STRING(255);
	(* Last values *)
	_lastValue			: STRING(255);
END_VAR

METHOD PROTECTED _handleVar
VAR_INPUT
END_VAR
IF NOT _isHmiConnected THEN RETURN; END_IF

(* Handle new messages *)
IF _Hmi.onNewMessage THEN
	IF (Tc2_Standard.FIND(STR1:= _Hmi.messageFullTopic, STR2:= _topicPrefix) <> 0) THEN
		IF (_Hmi.messageFullTopic = Tc2_Standard.CONCAT(STR1:= _topicPrefix, STR2:= 'value')) THEN
			_value:= _Hmi.messagePayload;
			_lastValue:= _value;
		END_IF
	END_IF
END_IF

(* Publish new messages *)
(* Value *)
IF (_lastValue <> _value) AND _timerPublish.Q THEN
	_lastValue:= _value;
	_Hmi.publish(
		topic	:= Tc2_Standard.CONCAT(STR1:= _topicPrefix, STR2:= 'value'),
		payload	:= _value);
END_IF
END_METHOD

METHOD FB_init : BOOL
VAR_INPUT
	bInitRetains	: BOOL; // if TRUE, the retain variables are initialized (warm start / cold start)
	bInCopyCode 	: BOOL;  // if TRUE, the instance afterwards gets moved into the copy code (online change)
	Hmi				: I_NexaHmi;
	id				: Tc2_System.T_MaxString;
	defaultValue	: STRING(255);
END_VAR
THIS^._value:= defaultValue;
END_METHOD

PROPERTY PUBLIC value : STRING(255)
GET
value:= _value;
END_GET
SET
_value:= value;
END_SET
END_PROPERTY

END_FUNCTION_BLOCK

// Persistent/FB_NexaHmiPersistentTIME
FUNCTION_BLOCK FB_NexaHmiPersistentTIME EXTENDS FB_NexaHmiPersistentBase
VAR
	_value				: TIME;
	(* Last values *)
	_lastValue			: TIME;
END_VAR

METHOD PROTECTED _handleVar
VAR_INPUT
END_VAR
IF NOT _isHmiConnected THEN RETURN; END_IF

(* Handle new messages *)
IF _Hmi.onNewMessage THEN
	IF (Tc2_Standard.FIND(STR1:= _Hmi.messageFullTopic, STR2:= _topicPrefix) <> 0) THEN
		IF (_Hmi.messageFullTopic = Tc2_Standard.CONCAT(STR1:= _topicPrefix, STR2:= 'value')) THEN
			_value:= UDINT_TO_TIME(STRING_TO_UDINT(_Hmi.messagePayload));
			_lastValue:= _value;
		END_IF
	END_IF
END_IF

(* Publish new messages *)
(* Value *)
IF (_lastValue <> _value) AND _timerPublish.Q THEN
	_lastValue:= _value;
	_Hmi.publish(
		topic	:= Tc2_Standard.CONCAT(STR1:= _topicPrefix, STR2:= 'value'),
		payload	:= UDINT_TO_STRING(TIME_TO_UDINT(_value)));
END_IF
END_METHOD

METHOD FB_init : BOOL
VAR_INPUT
	bInitRetains	: BOOL; // if TRUE, the retain variables are initialized (warm start / cold start)
	bInCopyCode 	: BOOL;  // if TRUE, the instance afterwards gets moved into the copy code (online change)
	Hmi				: I_NexaHmi;
	id				: Tc2_System.T_MaxString;
	defaultValue	: TIME;
END_VAR
THIS^._value:= defaultValue;
END_METHOD

PROPERTY PUBLIC value : TIME
GET
value:= _value;
END_GET
SET
_value:= value;
END_SET
END_PROPERTY

END_FUNCTION_BLOCK

// Persistent/FB_NexaHmiPersistentXYZ
FUNCTION_BLOCK FB_NexaHmiPersistentXYZ EXTENDS FB_NexaHmiPersistentBase
VAR
	_X					: REAL;
	_Y					: REAL;
	_Z					: REAL;
	_velocity			: REAL;
	(* General *)
	_payloadSplitter	: TcNexa_Components_TcUtilities.FB_TextSplitter;
	_tmpText			: Tc2_System.T_MaxString;
	(* Last values *)
	_lastX				: REAL;
	_lastY				: REAL;
	_lastZ				: REAL;
	_lastVelocity		: REAL;
END_VAR

METHOD PROTECTED _handleVar
VAR_INPUT
END_VAR
IF NOT _isHmiConnected THEN RETURN; END_IF

(* Handle new messages *)
IF _Hmi.onNewMessage THEN
	IF (Tc2_Standard.FIND(STR1:= _Hmi.messageFullTopic, STR2:= _topicPrefix) <> 0) THEN
		IF (_Hmi.messageFullTopic = Tc2_Standard.CONCAT(STR1:= _topicPrefix, STR2:= 'value')) THEN
			_payloadSplitter.split(
				source		:= _Hmi.messagePayload,
				delimiter	:= ';',
				Response	:= 0);
			_X:= STRING_TO_REAL(_payloadSplitter.getValueAt(index:= 1, Response:= 0));
			_lastX:= _X;
			_Y:= STRING_TO_REAL(_payloadSplitter.getValueAt(index:= 2, Response:= 0));
			_lastY:= _Y;
			_Z:= STRING_TO_REAL(_payloadSplitter.getValueAt(index:= 3, Response:= 0));
			_lastZ:= _Z;
			_velocity:= STRING_TO_REAL(_payloadSplitter.getValueAt(index:= 4, Response:= 0));
			_lastVelocity:= _velocity;
		END_IF
	END_IF
END_IF
(* Publish new messages *)
(* Value *)
IF ((_lastX <> _X) OR (_lastY <> _Y) OR (_lastZ <> _Z) OR (_lastVelocity <> _velocity)) AND _timerPublish.Q THEN
	_lastX:= _X;
	_lastY:= _Y;
	_lastZ:= _Z;
	_lastVelocity:= _velocity;
	_tmpText:= Tc2_Standard.CONCAT(
		STR1:= REAL_TO_STRING(_X),
		STR2:= ';');
	_tmpText:= Tc2_Standard.CONCAT(
		STR1:= _tmpText,
		STR2:= REAL_TO_STRING(_Y));
	_tmpText:= Tc2_Standard.CONCAT(
		STR1:= _tmpText,
		STR2:= ';');
	_tmpText:= Tc2_Standard.CONCAT(
		STR1:= _tmpText,
		STR2:= REAL_TO_STRING(_Z));
	_tmpText:= Tc2_Standard.CONCAT(
		STR1:= _tmpText,
		STR2:= ';');
	_tmpText:= Tc2_Standard.CONCAT(
		STR1:= _tmpText,
		STR2:= REAL_TO_STRING(_velocity));
	_tmpText:= Tc2_Standard.CONCAT(
		STR1:= _tmpText,
		STR2:= ';');
	_Hmi.publish(
		topic	:= Tc2_Standard.CONCAT(STR1:= _topicPrefix, STR2:= 'value'),
		payload	:= _tmpText);
END_IF
END_METHOD

METHOD FB_init : BOOL
VAR_INPUT
	bInitRetains		: BOOL; // if TRUE, the retain variables are initialized (warm start / cold start)
	bInCopyCode 		: BOOL;  // if TRUE, the instance afterwards gets moved into the copy code (online change)
	Hmi					: I_NexaHmi;
	id					: Tc2_System.T_MaxString;
	defaultX			: REAL;
	defaultY			: REAL;
	defaultZ			: REAL;
	defaultVelocity		: REAL;
END_VAR
THIS^._X:= defaultX;
THIS^._Y:= defaultY;
THIS^._Z:= defaultZ;
THIS^._velocity:= defaultVelocity;
END_METHOD

PROPERTY PUBLIC velocity : REAL
GET
velocity:= _velocity;
END_GET
SET
_velocity:= velocity;
END_SET
END_PROPERTY

PROPERTY PUBLIC X : REAL
GET
X:= _X;
END_GET
SET
_X:= X;
END_SET
END_PROPERTY

PROPERTY PUBLIC Y : REAL
GET
Y:= _Y;
END_GET
SET
_Y:= Y;
END_SET
END_PROPERTY

PROPERTY PUBLIC Z : REAL
GET
Z:= _Z;
END_GET
SET
_Z:= Z;
END_SET
END_PROPERTY

END_FUNCTION_BLOCK

// Settings/FB_NexaHmiSettingBase
FUNCTION_BLOCK ABSTRACT FB_NexaHmiSettingBase
VAR
	_Hmi				: I_NexaHmi;
	_onHmiConnection	: Tc2_Standard.R_TRIG;
	_isHmiConnected		: BOOL;
	_id					: UINT;
	_name				: STRING(255);
	_description		: STRING(255);
	_userLevel			: E_UserLevel:= E_UserLevel.Administrator;
	_enabled			: BOOL;
	(* General *)
	_timerPublish		: Tc2_Standard.TON;
	_dataReceived		: BOOL;
	_topicPrefix		: STRING(255);
	_lastEnabled		: BOOL;
	_lastUserLevel		: E_UserLevel;
END_VAR

METHOD PROTECTED ABSTRACT _handleVars
VAR_INPUT
END_VAR
END_METHOD

METHOD PROTECTED _onConnection
VAR_INPUT
END_VAR
IF NOT _onHmiConnection.Q THEN RETURN; END_IF

_topicPrefix:= Tc2_Standard.CONCAT(STR1:= _Hmi.topicPrefix, STR2:= _topicPrefix);
_topicPrefix:= Tc2_Standard.CONCAT(STR1:= _topicPrefix, STR2:= UINT_TO_STRING(_id));
_topicPrefix:= Tc2_Standard.CONCAT(STR1:= _topicPrefix, STR2:= '/');
_Hmi.subscribe(topic:= Tc2_Standard.CONCAT(STR1:= _topicPrefix, STR2:= 'value'));

_Hmi.publish(
	topic	:= Tc2_Standard.CONCAT(STR1:= _topicPrefix, STR2:= 'active'),
	payload	:= BOOL_TO_STRING(TRUE));
_Hmi.publish(
	topic	:= Tc2_Standard.CONCAT(STR1:= _topicPrefix, STR2:= 'name'),
	payload	:= _name);
_Hmi.publish(
	topic	:= Tc2_Standard.CONCAT(STR1:= _topicPrefix, STR2:= 'description'),
	payload	:= _description);
END_METHOD

METHOD PROTECTED _updateTopics
VAR_INPUT
END_VAR
IF NOT _isHmiConnected THEN RETURN; END_IF

(* Enabled *)
IF (_lastEnabled <> _enabled) OR _onHmiConnection.Q THEN
	_lastEnabled:= _enabled;
	_Hmi.publish(
		topic	:= Tc2_Standard.CONCAT(STR1:= _topicPrefix, STR2:= 'enabled'),
		payload	:= BOOL_TO_STRING(_enabled));
END_IF
(* User Level *)
IF (_lastUserLevel <> _userLevel) OR _onHmiConnection.Q THEN
	_lastUserLevel:= _userLevel;
	_Hmi.publish(
		topic	:= Tc2_Standard.CONCAT(STR1:= _topicPrefix, STR2:= 'userLevel'),
		payload	:= F_GetUserLevelAsString(userLevel:= _userLevel));
END_IF
END_METHOD

METHOD FB_init : BOOL
VAR_INPUT
	bInitRetains	: BOOL; // if TRUE, the retain variables are initialized (warm start / cold start)
	bInCopyCode 	: BOOL;  // if TRUE, the instance afterwards gets moved into the copy code (online change)
	Hmi				: I_NexaHmi;
	id				: UINT;
	name			: Tc2_System.T_MaxString;
	description		: Tc2_System.T_MaxString;
END_VAR
THIS^._Hmi:= Hmi;
THIS^._id:= id;
THIS^._name:= name;
THIS^._description:= description;
END_METHOD

PROPERTY description : Tc2_System.T_MaxString
GET
description:= _description;
END_GET
END_PROPERTY

PROPERTY enabled : BOOL
GET
enabled:= _enabled;
END_GET
SET
_enabled:= enabled;
END_SET
END_PROPERTY

PROPERTY name : Tc2_System.T_MaxString
GET
name:= _name;
END_GET
END_PROPERTY

PROPERTY userLevel : E_UserLevel
GET
userLevel:= _userLevel;
END_GET
SET
_userLevel:= userLevel;
END_SET
END_PROPERTY

METHOD PUBLIC FB_main
VAR_INPUT
END_VAR
_timerPublish(
	IN	:= _isHmiConnected AND NOT _dataReceived, 
	PT	:= T#1S);
_isHmiConnected:= _Hmi.isConnected;
_onHmiConnection(CLK:= _isHmiConnected);

_onConnection();
_updateTopics();
_handleVars();
END_METHOD

END_FUNCTION_BLOCK

// Settings/FB_NexaHmiSettingBOOL
FUNCTION_BLOCK FB_NexaHmiSettingBOOL EXTENDS FB_NexaHmiSettingBase
VAR
	_value				: BOOL;
END_VAR

METHOD PROTECTED _handleVars
VAR_INPUT
END_VAR
IF NOT _isHmiConnected THEN RETURN; END_IF

(* Handle new messages *)
IF _Hmi.onNewMessage THEN
	IF (Tc2_Standard.FIND(STR1:= _Hmi.messageFullTopic, STR2:= _topicPrefix) <> 0) THEN
		IF (_Hmi.messageFullTopic = Tc2_Standard.CONCAT(STR1:= _topicPrefix, STR2:= 'value')) THEN
			_value:= STRING_TO_BOOL(_Hmi.messagePayload);
			_dataReceived:= TRUE;
		END_IF
	END_IF
END_IF

(* Publish new messages *)
(* Value *)
IF _timerPublish.Q THEN
	_dataReceived:= TRUE;
	_Hmi.publish(
		topic	:= Tc2_Standard.CONCAT(STR1:= _topicPrefix, STR2:= 'value'),
		payload	:= BOOL_TO_STRING(_value));
END_IF
END_METHOD

METHOD FB_init : BOOL
VAR_INPUT
	bInitRetains	: BOOL; // if TRUE, the retain variables are initialized (warm start / cold start)
	bInCopyCode 	: BOOL;  // if TRUE, the instance afterwards gets moved into the copy code (online change)
	Hmi				: I_NexaHmi;
	id				: UINT;
	name			: Tc2_System.T_MaxString;
	description		: Tc2_System.T_MaxString;
	defaultValue	: BOOL;
END_VAR
THIS^._value:= defaultValue;

_topicPrefix:= 'settings/booleans/';
END_METHOD

PROPERTY PUBLIC value : BOOL
GET
value:= _value;
END_GET
END_PROPERTY

END_FUNCTION_BLOCK

// Settings/FB_NexaHmiSettingCHOICE
FUNCTION_BLOCK FB_NexaHmiSettingCHOICE EXTENDS FB_NexaHmiSettingBase
VAR
	_choices			: STRING(255);	
	_value				: STRING(255);
	(* Last values *)
	_Splitter			: TcNexa_Components_TcUtilities.FB_TextSplitter;
END_VAR

METHOD PROTECTED _handleVars
VAR_INPUT
END_VAR
IF NOT _isHmiConnected THEN RETURN; END_IF

(* Handle new messages *)
IF _Hmi.onNewMessage THEN
	IF (Tc2_Standard.FIND(STR1:= _Hmi.messageFullTopic, STR2:= _topicPrefix) <> 0) THEN
		IF (_Hmi.messageFullTopic = Tc2_Standard.CONCAT(STR1:= _topicPrefix, STR2:= 'value')) THEN
			_value:= _Hmi.messagePayload;
			_dataReceived:= TRUE;
		END_IF
	END_IF
END_IF

(* Publish new messages *)
IF _onHmiConnection.Q THEN
	_Hmi.publish(
		topic	:= Tc2_Standard.CONCAT(STR1:= _topicPrefix, STR2:= 'choices'),
		payload	:= _choices);	
END_IF
(* Value *)
IF _timerPublish.Q THEN
	_dataReceived:= TRUE;
	_Hmi.publish(
		topic	:= Tc2_Standard.CONCAT(STR1:= _topicPrefix, STR2:= 'value'),
		payload	:= _value);
END_IF
END_METHOD

METHOD FB_init : BOOL
VAR_INPUT
	bInitRetains	: BOOL; // if TRUE, the retain variables are initialized (warm start / cold start)
	bInCopyCode 	: BOOL;  // if TRUE, the instance afterwards gets moved into the copy code (online change)
	Hmi				: I_NexaHmi;
	id				: UINT;
	name			: STRING(255);
	description		: STRING(255);
	choices			: STRING(255);	// List of string as choices with delimiter ","
END_VAR
_Splitter.split(
	source		:= choices,
	delimiter	:= ',',
	Response	:= 0);

THIS^._choices:= choices;
THIS^._value:= _Splitter.getValueAt(1, 0);
_topicPrefix:= 'settings/choices/';
END_METHOD

PROPERTY PUBLIC value : STRING(255)
GET
value:= _value;
END_GET
END_PROPERTY

END_FUNCTION_BLOCK

// Settings/FB_NexaHmiSettingINT
FUNCTION_BLOCK FB_NexaHmiSettingINT EXTENDS FB_NexaHmiSettingBase
VAR
	_value				: INT;
	_lowerLimit			: INT:= -32768;
	_hasLowerLimit		: BOOL;
	_upperLimit			: INT:= 32767;
	_hasUpperLimit		: BOOL;
END_VAR

METHOD PROTECTED _handleVars
VAR_INPUT
END_VAR
IF NOT _isHmiConnected THEN RETURN; END_IF

(* Handle new messages *)
IF _Hmi.onNewMessage THEN
	IF (Tc2_Standard.FIND(STR1:= _Hmi.messageFullTopic, STR2:= _topicPrefix) <> 0) THEN
		IF (_Hmi.messageFullTopic = Tc2_Standard.CONCAT(STR1:= _topicPrefix, STR2:= 'value')) THEN
			_value:= STRING_TO_INT(_Hmi.messagePayload);
			_dataReceived:= TRUE;
		END_IF
	END_IF
END_IF

(* Publish new messages *)
(* Value *)
IF _timerPublish.Q THEN
	_dataReceived:= TRUE;
	_Hmi.publish(
		topic	:= Tc2_Standard.CONCAT(STR1:= _topicPrefix, STR2:= 'value'),
		payload	:= INT_TO_STRING(_value));
END_IF

(* Publish only on connection *)
IF NOT _onHmiConnection.Q THEN RETURN; END_IF

(* Upper Value *)
IF _hasLowerLimit THEN
	_Hmi.publish(
		topic	:= Tc2_Standard.CONCAT(STR1:= _topicPrefix, STR2:= 'min'),
		payload	:= INT_TO_STRING(_lowerLimit));
END_IF
(* Lower Value *)
IF _hasUpperLimit THEN
	_Hmi.publish(
		topic	:= Tc2_Standard.CONCAT(STR1:= _topicPrefix, STR2:= 'max'),
		payload	:= INT_TO_STRING(_upperLimit));
END_IF
END_METHOD

METHOD FB_init : BOOL
VAR_INPUT
	bInitRetains	: BOOL; // if TRUE, the retain variables are initialized (warm start / cold start)
	bInCopyCode 	: BOOL;  // if TRUE, the instance afterwards gets moved into the copy code (online change)
	Hmi				: I_NexaHmi;
	id				: UINT;
	name			: Tc2_System.T_MaxString;
	description		: Tc2_System.T_MaxString;
	defaultValue	: INT;
	lowerLimit		: INT;
	hasLowerLimit	: BOOL;
	upperLimit		: INT;
	hasUpperLimit	: BOOL;
END_VAR
THIS^._value:= defaultValue;
THIS^._lowerLimit:= lowerLimit;
THIS^._hasLowerLimit:= hasLowerLimit;
THIS^._upperLimit:= upperLimit;
THIS^._hasUpperLimit:= hasUpperLimit;

_topicPrefix:= 'settings/integers/';
END_METHOD

PROPERTY PUBLIC lowerLimit : INT
GET
lowerLimit:= _lowerLimit;
END_GET
END_PROPERTY

PROPERTY PUBLIC upperLimit : INT
GET
upperLimit:= _upperLimit;
END_GET
END_PROPERTY

PROPERTY PUBLIC value : INT
GET
value:= _value;
END_GET
END_PROPERTY

END_FUNCTION_BLOCK

// Settings/FB_NexaHmiSettingREAL
FUNCTION_BLOCK FB_NexaHmiSettingREAL EXTENDS FB_NexaHmiSettingBase
VAR
	_value				: REAL;
	_lowerLimit			: REAL:= -3.402823E+38;
	_hasLowerLimit		: BOOL;
	_upperLimit			: REAL:= 3.402823E+38;
	_hasUpperLimit		: BOOL;
	_unit				: STRING;
END_VAR

METHOD PROTECTED _handleVars
VAR_INPUT
END_VAR
IF NOT _isHmiConnected THEN RETURN; END_IF

(* Handle new messages *)
IF _Hmi.onNewMessage THEN
	IF (Tc2_Standard.FIND(STR1:= _Hmi.messageFullTopic, STR2:= _topicPrefix) <> 0) THEN
		IF (_Hmi.messageFullTopic = Tc2_Standard.CONCAT(STR1:= _topicPrefix, STR2:= 'value')) THEN
			_value:= STRING_TO_REAL(_Hmi.messagePayload);
			_dataReceived:= TRUE;
		END_IF
	END_IF
END_IF

(* Publish new messages *)
(* Value *)
IF _timerPublish.Q THEN
	_dataReceived:= TRUE;
	_Hmi.publish(
		topic	:= Tc2_Standard.CONCAT(STR1:= _topicPrefix, STR2:= 'value'),
		payload	:= REAL_TO_STRING(_value));
END_IF

(* Publish only on connection *)
IF NOT _onHmiConnection.Q THEN RETURN; END_IF

(* Unit *)
_Hmi.publish(
	topic	:= Tc2_Standard.CONCAT(STR1:= _topicPrefix, STR2:= 'unit'),
	payload	:= _unit);
(* Upper Limit *)
IF _hasLowerLimit THEN
	_Hmi.publish(
		topic	:= Tc2_Standard.CONCAT(STR1:= _topicPrefix, STR2:= 'min'),
		payload	:= REAL_TO_STRING(_lowerLimit));
END_IF
(* Lower Limit *)
IF _hasUpperLimit THEN
	_Hmi.publish(
		topic	:= Tc2_Standard.CONCAT(STR1:= _topicPrefix, STR2:= 'max'),
		payload	:= REAL_TO_STRING(_upperLimit));
END_IF
END_METHOD

METHOD FB_init : BOOL
VAR_INPUT
	bInitRetains	: BOOL; // if TRUE, the retain variables are initialized (warm start / cold start)
	bInCopyCode 	: BOOL;  // if TRUE, the instance afterwards gets moved into the copy code (online change)
	Hmi				: I_NexaHmi;
	id				: UINT;
	name			: Tc2_System.T_MaxString;
	description		: Tc2_System.T_MaxString;
	defaultValue	: REAL;
	lowerLimit		: REAL;
	hasLowerLimit	: BOOL;
	upperLimit		: REAL;
	hasUpperLimit	: BOOL;
	unit			: STRING;
END_VAR
THIS^._value:= defaultValue;
THIS^._lowerLimit:= lowerLimit;
THIS^._hasLowerLimit:= hasLowerLimit;
THIS^._upperLimit:= upperLimit;
THIS^._hasUpperLimit:= hasUpperLimit;
THIS^._unit:= unit;

_topicPrefix:= 'settings/reals/';
END_METHOD

PROPERTY PUBLIC lowerLimit : REAL
GET
lowerLimit:= _lowerLimit;
END_GET
END_PROPERTY

PROPERTY PUBLIC upperLimit : REAL
GET
upperLimit:= _upperLimit;
END_GET
END_PROPERTY

PROPERTY PUBLIC value : REAL
GET
value:= _value;
END_GET
END_PROPERTY

END_FUNCTION_BLOCK

// Settings/FB_NexaHmiSettingSTRING
FUNCTION_BLOCK FB_NexaHmiSettingSTRING EXTENDS FB_NexaHmiSettingBase
VAR
	_value				: STRING(255);
END_VAR

METHOD PROTECTED _handleVars
VAR_INPUT
END_VAR
IF NOT _isHmiConnected THEN RETURN; END_IF

(* Handle new messages *)
IF _Hmi.onNewMessage THEN
	IF (Tc2_Standard.FIND(STR1:= _Hmi.messageFullTopic, STR2:= _topicPrefix) <> 0) THEN
		IF (_Hmi.messageFullTopic = Tc2_Standard.CONCAT(STR1:= _topicPrefix, STR2:= 'value')) THEN
			_value:= _Hmi.messagePayload;
			_dataReceived:= TRUE;
		END_IF
	END_IF
END_IF

(* Publish new messages *)
(* Value *)
IF _timerPublish.Q THEN
	_dataReceived:= TRUE;
	_Hmi.publish(
		topic	:= Tc2_Standard.CONCAT(STR1:= _topicPrefix, STR2:= 'value'),
		payload	:= _value);
END_IF
END_METHOD

METHOD FB_init : BOOL
VAR_INPUT
	bInitRetains	: BOOL; // if TRUE, the retain variables are initialized (warm start / cold start)
	bInCopyCode 	: BOOL;  // if TRUE, the instance afterwards gets moved into the copy code (online change)
	Hmi				: I_NexaHmi;
	id				: UINT;
	name			: Tc2_System.T_MaxString;
	description		: Tc2_System.T_MaxString;
	defaultValue	: Tc2_System.T_MaxString;
END_VAR
THIS^._value:= defaultValue;
_topicPrefix:= 'settings/strings/';
END_METHOD

PROPERTY PUBLIC value : STRING(255)
GET
value:= _value;
END_GET
END_PROPERTY

END_FUNCTION_BLOCK

// Settings/FB_NexaHmiSettingTIME
FUNCTION_BLOCK FB_NexaHmiSettingTIME EXTENDS FB_NexaHmiSettingBase
VAR
	_value				: TIME;
	_lowerLimit			: TIME;
	_hasLowerLimit		: BOOL;
	_upperLimit			: TIME;
	_hasUpperLimit		: BOOL;
END_VAR

METHOD PROTECTED _handleVars
VAR_INPUT
END_VAR
IF NOT _isHmiConnected THEN RETURN; END_IF

(* Handle new messages *)
IF _Hmi.onNewMessage THEN
	IF (Tc2_Standard.FIND(STR1:= _Hmi.messageFullTopic, STR2:= _topicPrefix) <> 0) THEN
		IF (_Hmi.messageFullTopic = Tc2_Standard.CONCAT(STR1:= _topicPrefix, STR2:= 'value')) THEN
			_value:= UDINT_TO_TIME(STRING_TO_UDINT(_Hmi.messagePayload));
			_dataReceived:= TRUE;
		END_IF
	END_IF
END_IF

(* Publish new messages *)
(* Value *)
IF _timerPublish.Q THEN
	_dataReceived:= TRUE;
	_Hmi.publish(
		topic	:= Tc2_Standard.CONCAT(STR1:= _topicPrefix, STR2:= 'value'),
		payload	:= UDINT_TO_STRING(TIME_TO_UDINT(_value)));
END_IF

(* Publish only on connection *)
IF NOT _onHmiConnection.Q THEN RETURN; END_IF

(* Upper Limit *)
IF _hasLowerLimit THEN
	_Hmi.publish(
		topic	:= Tc2_Standard.CONCAT(STR1:= _topicPrefix, STR2:= 'min'),
		payload	:= UDINT_TO_STRING(TIME_TO_UDINT(_lowerLimit)));
END_IF
(* Lower Limit *)
IF _hasUpperLimit THEN
	_Hmi.publish(
		topic	:= Tc2_Standard.CONCAT(STR1:= _topicPrefix, STR2:= 'max'),
		payload	:= UDINT_TO_STRING(TIME_TO_UDINT(_upperLimit)));
END_IF
END_METHOD

METHOD FB_init : BOOL
VAR_INPUT
	bInitRetains	: BOOL; // if TRUE, the retain variables are initialized (warm start / cold start)
	bInCopyCode 	: BOOL;  // if TRUE, the instance afterwards gets moved into the copy code (online change)
	Hmi				: I_NexaHmi;
	id				: UINT;
	name			: Tc2_System.T_MaxString;
	description		: Tc2_System.T_MaxString;
	defaultValue	: TIME;
	lowerLimit		: TIME;
	hasLowerLimit	: BOOL;
	upperLimit		: TIME;
	hasUpperLimit	: BOOL;
END_VAR
THIS^._value:= defaultValue;
THIS^._lowerLimit:= lowerLimit;
THIS^._hasLowerLimit:= hasLowerLimit;
THIS^._upperLimit:= upperLimit;
THIS^._hasUpperLimit:= hasUpperLimit;

_topicPrefix:= 'settings/times/';
END_METHOD

PROPERTY PUBLIC lowerLimit : TIME
GET
lowerLimit:= _lowerLimit;
END_GET
END_PROPERTY

PROPERTY PUBLIC upperLimit : TIME
GET
upperLimit:= _upperLimit;
END_GET
END_PROPERTY

PROPERTY PUBLIC value : TIME
GET
value:= _value;
END_GET
END_PROPERTY

END_FUNCTION_BLOCK

// Tests/PRG_TEST
PROGRAM PRG_TEST
VAR
	_test : FB_NexaHmi;
END_VAR

END_PROGRAM
